LIN {X 0,Y 525.291,Z 461.786,A -85,B 0,C 180,E1 -4783.393,E2 -4783.393} C_VEL
LIN {X 0,Y 525.461,Z 449.021,A -85,B 0,C 180,E1 -4783.659,E2 -4783.659} C_VEL
LIN {X 0,Y 525.774,Z 355.172,A -85,B 0,C 180,E1 -4784.965,E2 -4784.965} C_VEL
LIN {X 0,Y 524.31,Z 344.888,A -85,B 0,C 180,E1 -4785.179,E2 -4785.179} C_VEL
LIN {X 0,Y 524.712,Z 325.315,A -85,B 0,C 180,E1 -4788.014,E2 -4788.014} C_VEL
LIN {X 0,Y 525.255,Z 302.194,A -85,B 0,C 180,E1 -4791.383,E2 -4791.383} C_VEL
LIN {X 0,Y 525.641,Z 284.25,A -85,B 0,C 180,E1 -4794.065,E2 -4794.065} C_VEL
LIN {X 0,Y 523.939,Z 275.222,A -85,B 0,C 180,E1 -4795.549,E2 -4795.549} C_VEL
LIN {X 0,Y 523.92,Z 275.224,A -85,B 0,C 180,E1 -4798.874,E2 -4798.874} C_VEL
LIN {X 0,Y 523.911,Z 275.22,A -85,B 0,C 180,E1 -4801.543,E2 -4801.543} C_VEL
LIN {X 0,Y 523.903,Z 275.225,A -85,B 0,C 180,E1 -4804.29,E2 -4804.29} C_VEL
LIN {X 0,Y 523.871,Z 275.227,A -85,B 0,C 180,E1 -4807.132,E2 -4807.132} C_VEL
LIN {X 0,Y 523.9,Z 275.223,A -85,B 0,C 180,E1 -4810.124,E2 -4810.124} C_VEL
LIN {X 0,Y 523.873,Z 275.226,A -85,B 0,C 180,E1 -4813.168,E2 -4813.168} C_VEL
LIN {X 0,Y 523.907,Z 275.22,A -85,B 0,C 180,E1 -4815.768,E2 -4815.768} C_VEL
LIN {X 0,Y 523.878,Z 275.229,A -85,B 0,C 180,E1 -4818.901,E2 -4818.901} C_VEL
LIN {X 0,Y 523.887,Z 275.223,A -85,B 0,C 180,E1 -4821.895,E2 -4821.895} C_VEL
LIN {X 0,Y 523.895,Z 275.228,A -85,B 0,C 180,E1 -4824.91,E2 -4824.91} C_VEL
LIN {X 0,Y 523.906,Z 275.22,A -85,B 0,C 180,E1 -4827.678,E2 -4827.678} C_VEL
LIN {X 0,Y 523.921,Z 275.226,A -85,B 0,C 180,E1 -4830.675,E2 -4830.675} C_VEL
LIN {X 0,Y 523.909,Z 275.227,A -85,B 0,C 180,E1 -4832.864,E2 -4832.864} C_VEL
LIN {X 0,Y 523.899,Z 275.222,A -85,B 0,C 180,E1 -4835.802,E2 -4835.802} C_VEL
LIN {X 0,Y 523.907,Z 275.228,A -85,B 0,C 180,E1 -4838.765,E2 -4838.765} C_VEL
LIN {X 0,Y 523.902,Z 275.224,A -85,B 0,C 180,E1 -4841.219,E2 -4841.219} C_VEL
LIN {X 0,Y 523.89,Z 275.223,A -85,B 0,C 180,E1 -4843.637,E2 -4843.637} C_VEL
LIN {X 0,Y 523.894,Z 275.223,A -85,B 0,C 180,E1 -4846.026,E2 -4846.026} C_VEL
LIN {X 0,Y 523.975,Z 275.216,A -85,B 0,C 180,E1 -4848.393,E2 -4848.393} C_VEL
LIN {X 0,Y 523.964,Z 275.214,A -85,B 0,C 180,E1 -4851.515,E2 -4851.515} C_VEL
LIN {X 0,Y 524.043,Z 275.21,A -85,B 0,C 180,E1 -4854.613,E2 -4854.613} C_VEL
LIN {X 0,Y 524.066,Z 275.201,A -85,B 0,C 180,E1 -4857.694,E2 -4857.694} C_VEL
LIN {X 0,Y 524.089,Z 275.205,A -85,B 0,C 180,E1 -4860.768,E2 -4860.768} C_VEL
LIN {X 0,Y 524.037,Z 275.21,A -85,B 0,C 180,E1 -4863.075,E2 -4863.075} C_VEL
LIN {X 0,Y 523.997,Z 275.211,A -85,B 0,C 180,E1 -4866.159,E2 -4866.159} C_VEL
LIN {X 0,Y 523.969,Z 275.216,A -85,B 0,C 180,E1 -4869.262,E2 -4869.262} C_VEL
LIN {X 0,Y 523.986,Z 275.211,A -85,B 0,C 180,E1 -4871.752,E2 -4871.752} C_VEL
LIN {X 0,Y 523.954,Z 275.222,A -85,B 0,C 180,E1 -4875.053,E2 -4875.053} C_VEL
LIN {X 0,Y 523.928,Z 275.219,A -85,B 0,C 180,E1 -4877.97,E2 -4877.97} C_VEL
LIN {X 0,Y 523.937,Z 275.22,A -85,B 0,C 180,E1 -4880.411,E2 -4880.411} C_VEL
LIN {X 0,Y 523.881,Z 275.23,A -85,B 0,C 180,E1 -4882.894,E2 -4882.894} C_VEL
LIN {X 0,Y 523.92,Z 275.222,A -85,B 0,C 180,E1 -4885.42,E2 -4885.42} C_VEL
LIN {X 0,Y 523.939,Z 275.217,A -85,B 0,C 180,E1 -4888,E2 -4888} C_VEL
LIN {X 0,Y 523.922,Z 275.225,A -85,B 0,C 180,E1 -4890.858,E2 -4890.858} C_VEL
LIN {X 0,Y 523.934,Z 275.218,A -85,B 0,C 180,E1 -4893.737,E2 -4893.737} C_VEL
LIN {X 0,Y 523.897,Z 275.225,A -85,B 0,C 180,E1 -4896.406,E2 -4896.406} C_VEL
LIN {X 0,Y 523.934,Z 275.224,A -85,B 0,C 180,E1 -4899.083,E2 -4899.083} C_VEL
LIN {X 0,Y 523.934,Z 275.218,A -85,B 0,C 180,E1 -4902.12,E2 -4902.12} C_VEL
LIN {X 0,Y 523.935,Z 275.222,A -85,B 0,C 180,E1 -4905.31,E2 -4905.31} C_VEL
LIN {X 0,Y 523.903,Z 275.227,A -85,B 0,C 180,E1 -4906.94,E2 -4906.94} C_VEL
LIN {X 0,Y 523.24,Z 275.307,A -85,B 0,C 180,E1 -4907.581,E2 -4907.581} C_VEL
LIN {X 0,Y 520.405,Z 275.662,A -85,B 0,C 180,E1 -4908.623,E2 -4908.623} C_VEL
LIN {X 0,Y 518.008,Z 275.959,A -85,B 0,C 180,E1 -4909.462,E2 -4909.462} C_VEL
LIN {X 0,Y 516.978,Z 276.085,A -85,B 0,C 180,E1 -4910.11,E2 -4910.11} C_VEL
LIN {X 0,Y 516.894,Z 276.096,A -85,B 0,C 180,E1 -4910.33,E2 -4910.33} C_VEL
LIN {X 0,Y 516.872,Z 276.101,A -85,B 0,C 180,E1 -4913.343,E2 -4913.343} C_VEL
LIN {X 0,Y 516.898,Z 276.094,A -85,B 0,C 180,E1 -4916.122,E2 -4916.122} C_VEL
LIN {X 0,Y 516.88,Z 276.103,A -85,B 0,C 180,E1 -4918.937,E2 -4918.937} C_VEL
LIN {X 0,Y 516.911,Z 276.094,A -85,B 0,C 180,E1 -4921.586,E2 -4921.586} C_VEL
LIN {X 0,Y 516.923,Z 276.091,A -85,B 0,C 180,E1 -4924.212,E2 -4924.212} C_VEL
LIN {X 0,Y 516.858,Z 276.105,A -85,B 0,C 180,E1 -4926.777,E2 -4926.777} C_VEL
LIN {X 0,Y 516.934,Z 276.09,A -85,B 0,C 180,E1 -4929.732,E2 -4929.732} C_VEL
LIN {X 0,Y 516.925,Z 276.094,A -85,B 0,C 180,E1 -4932.597,E2 -4932.597} C_VEL
LIN {X 0,Y 516.939,Z 276.095,A -85,B 0,C 180,E1 -4935.03,E2 -4935.03} C_VEL
LIN {X 0,Y 516.963,Z 276.086,A -85,B 0,C 180,E1 -4938.234,E2 -4938.234} C_VEL
LIN {X 0,Y 516.967,Z 276.09,A -85,B 0,C 180,E1 -4941.399,E2 -4941.399} C_VEL
LIN {X 0,Y 517.008,Z 276.081,A -85,B 0,C 180,E1 -4943.756,E2 -4943.756} C_VEL
LIN {X 0,Y 517.083,Z 276.073,A -85,B 0,C 180,E1 -4947.662,E2 -4947.662} C_VEL
LIN {X 0,Y 517.09,Z 276.074,A -85,B 0,C 180,E1 -4950.777,E2 -4950.777} C_VEL
LIN {X 0,Y 517.011,Z 276.087,A -85,B 0,C 180,E1 -4953.115,E2 -4953.115} C_VEL
LIN {X 0,Y 516.998,Z 276.081,A -85,B 0,C 180,E1 -4956.241,E2 -4956.241} C_VEL
LIN {X 0,Y 516.947,Z 276.092,A -85,B 0,C 180,E1 -4959.387,E2 -4959.387} C_VEL
LIN {X 0,Y 516.977,Z 276.085,A -85,B 0,C 180,E1 -4961.822,E2 -4961.822} C_VEL
LIN {X 0,Y 516.935,Z 276.096,A -85,B 0,C 180,E1 -4965.144,E2 -4965.144} C_VEL
LIN {X 0,Y 516.915,Z 276.091,A -85,B 0,C 180,E1 -4968.219,E2 -4968.219} C_VEL
LIN {X 0,Y 516.903,Z 276.095,A -85,B 0,C 180,E1 -4970.698,E2 -4970.698} C_VEL
LIN {X 0,Y 516.877,Z 276.103,A -85,B 0,C 180,E1 -4973.219,E2 -4973.219} C_VEL
LIN {X 0,Y 516.928,Z 276.089,A -85,B 0,C 180,E1 -4976.194,E2 -4976.194} C_VEL
LIN {X 0,Y 516.916,Z 276.098,A -85,B 0,C 180,E1 -4979.3,E2 -4979.3} C_VEL
LIN {X 0,Y 516.881,Z 276.096,A -85,B 0,C 180,E1 -4982.541,E2 -4982.541} C_VEL
LIN {X 0,Y 516.858,Z 276.105,A -85,B 0,C 180,E1 -4985.329,E2 -4985.329} C_VEL
LIN {X 0,Y 516.858,Z 276.098,A -85,B 0,C 180,E1 -4987.941,E2 -4987.941} C_VEL
LIN {X 0,Y 516.886,Z 276.098,A -85,B 0,C 180,E1 -4990.735,E2 -4990.735} C_VEL
LIN {X 0,Y 517.02,Z 276.175,A -85,B 0,C 180,E1 -4993.84,E2 -4993.84} C_VEL
LIN {X 0,Y 517.32,Z 280.633,A -85,B 0,C 180,E1 -4994.754,E2 -4994.754} C_VEL
LIN {X 0,Y 517.177,Z 290.379,A -85,B 0,C 180,E1 -4996.7,E2 -4996.7} C_VEL
LIN {X 0,Y 519.112,Z 300.838,A -85,B 0,C 180,E1 -4996.916,E2 -4996.916} C_VEL
LIN {X 0,Y 518.557,Z 397.529,A -85,B 0,C 180,E1 -4998.312,E2 -4998.312} C_VEL
LIN {X 0,Y 518.413,Z 410.717,A -85,B 0,C 180,E1 -4998.665,E2 -4998.665} C_VEL
LIN {X 0,Y 518.158,Z 422.479,A -85,B 0,C 180,E1 -4999.124,E2 -4999.124} C_VEL
LIN {X 0,Y 517.938,Z 434.251,A -85,B 0,C 180,E1 -4999.742,E2 -4999.742} C_VEL
LIN {X 0,Y 517.615,Z 444.905,A -85,B 0,C 180,E1 -5000.459,E2 -5000.459} C_VEL
LIN {X 0,Y 517.342,Z 455.25,A -85,B 0,C 180,E1 -5001.326,E2 -5001.326} C_VEL
LIN {X 0,Y 517.089,Z 464.659,A -85,B 0,C 180,E1 -5002.294,E2 -5002.294} C_VEL
LIN {X 0,Y 516.852,Z 472.928,A -85,B 0,C 180,E1 -5003.337,E2 -5003.337} C_VEL
LIN {X 0,Y 516.659,Z 480.32,A -85,B 0,C 180,E1 -5004.488,E2 -5004.488} C_VEL
LIN {X 0,Y 516.517,Z 486.204,A -85,B 0,C 180,E1 -5005.621,E2 -5005.621} C_VEL
LIN {X 0,Y 516.373,Z 491.862,A -85,B 0,C 180,E1 -5007.016,E2 -5007.016} C_VEL
LIN {X 0,Y 516.34,Z 495.956,A -85,B 0,C 180,E1 -5008.398,E2 -5008.398} C_VEL
LIN {X 0,Y 516.238,Z 498.614,A -85,B 0,C 180,E1 -5009.755,E2 -5009.755} C_VEL
LIN {X 0,Y 516.205,Z 499.695,A -85,B 0,C 180,E1 -5010.651,E2 -5010.651} C_VEL
LIN {X 0,Y 516.199,Z 500.248,A -85,B 0,C 180,E1 -5011.542,E2 -5011.542} C_VEL
LIN {X 0,Y 516.168,Z 500.291,A -85,B 0,C 180,E1 -5012.424,E2 -5012.424} C_VEL
LIN {X 0,Y 516.187,Z 499.855,A -85,B 0,C 180,E1 -5013.302,E2 -5013.302} C_VEL
LIN {X 0,Y 516.226,Z 498.881,A -85,B 0,C 180,E1 -5014.174,E2 -5014.174} C_VEL
LIN {X 0,Y 516.272,Z 497.427,A -85,B 0,C 180,E1 -5015.039,E2 -5015.039} C_VEL
LIN {X 0,Y 516.4,Z 494.312,A -85,B 0,C 180,E1 -5016.33,E2 -5016.33} C_VEL
LIN {X 0,Y 516.455,Z 489.615,A -85,B 0,C 180,E1 -5017.704,E2 -5017.704} C_VEL
LIN {X 0,Y 516.569,Z 483.336,A -85,B 0,C 180,E1 -5019.076,E2 -5019.076} C_VEL
LIN {X 0,Y 516.801,Z 475.952,A -85,B 0,C 180,E1 -5020.332,E2 -5020.332} C_VEL
LIN {X 0,Y 516.981,Z 468.38,A -85,B 0,C 180,E1 -5021.37,E2 -5021.37} C_VEL
LIN {X 0,Y 517.287,Z 458.631,A -85,B 0,C 180,E1 -5022.455,E2 -5022.455} C_VEL
LIN {X 0,Y 517.533,Z 448.953,A -85,B 0,C 180,E1 -5023.33,E2 -5023.33} C_VEL
LIN {X 0,Y 517.863,Z 437.568,A -85,B 0,C 180,E1 -5024.15,E2 -5024.15} C_VEL
LIN {X 0,Y 518.14,Z 425.417,A -85,B 0,C 180,E1 -5024.832,E2 -5024.832} C_VEL
LIN {X 0,Y 518.303,Z 413.887,A -85,B 0,C 180,E1 -5025.322,E2 -5025.322} C_VEL
LIN {X 0,Y 518.48,Z 401.522,A -85,B 0,C 180,E1 -5025.69,E2 -5025.69} C_VEL
LIN {X 0,Y 518.625,Z 386.132,A -85,B 0,C 180,E1 -5025.957,E2 -5025.957} C_VEL
LIN {X 0,Y 519.014,Z 299.941,A -85,B 0,C 180,E1 -5027.195,E2 -5027.195} C_VEL
LIN {X 0,Y 517.1,Z 289.663,A -85,B 0,C 180,E1 -5027.42,E2 -5027.42} C_VEL
LIN {X 0,Y 516.929,Z 276.096,A -85,B 0,C 180,E1 -5029.622,E2 -5029.622} C_VEL
LIN {X 0,Y 516.953,Z 276.095,A -85,B 0,C 180,E1 -5032.972,E2 -5032.972} C_VEL
LIN {X 0,Y 516.877,Z 276.102,A -85,B 0,C 180,E1 -5035.321,E2 -5035.321} C_VEL
LIN {X 0,Y 517.021,Z 276.081,A -85,B 0,C 180,E1 -5037.663,E2 -5037.663} C_VEL
LIN {X 0,Y 517.038,Z 276.083,A -85,B 0,C 180,E1 -5040.779,E2 -5040.779} C_VEL
LIN {X 0,Y 516.987,Z 276.09,A -85,B 0,C 180,E1 -5043.117,E2 -5043.117} C_VEL
LIN {X 0,Y 516.95,Z 276.088,A -85,B 0,C 180,E1 -5046.244,E2 -5046.244} C_VEL
LIN {X 0,Y 516.906,Z 276.096,A -85,B 0,C 180,E1 -5049.39,E2 -5049.39} C_VEL
LIN {X 0,Y 516.925,Z 276.09,A -85,B 0,C 180,E1 -5051.826,E2 -5051.826} C_VEL
LIN {X 0,Y 516.899,Z 276.1,A -85,B 0,C 180,E1 -5055.154,E2 -5055.154} C_VEL
LIN {X 0,Y 516.872,Z 276.095,A -85,B 0,C 180,E1 -5058.225,E2 -5058.225} C_VEL
LIN {X 0,Y 516.859,Z 276.1,A -85,B 0,C 180,E1 -5060.704,E2 -5060.704} C_VEL
LIN {X 0,Y 516.86,Z 276.098,A -85,B 0,C 180,E1 -5064.075,E2 -5064.075} C_VEL
LIN {X 0,Y 516.88,Z 276.096,A -85,B 0,C 180,E1 -5066.661,E2 -5066.661} C_VEL
LIN {X 0,Y 516.863,Z 276.101,A -85,B 0,C 180,E1 -5069.527,E2 -5069.527} C_VEL
LIN {X 0,Y 516.856,Z 276.099,A -85,B 0,C 180,E1 -5072.548,E2 -5072.548} C_VEL
LIN {X 0,Y 516.84,Z 276.108,A -85,B 0,C 180,E1 -5075.336,E2 -5075.336} C_VEL
LIN {X 0,Y 516.841,Z 276.101,A -85,B 0,C 180,E1 -5077.947,E2 -5077.947} C_VEL
LIN {X 0,Y 516.872,Z 276.098,A -85,B 0,C 180,E1 -5080.743,E2 -5080.743} C_VEL
LIN {X 0,Y 516.849,Z 276.1,A -85,B 0,C 180,E1 -5083.907,E2 -5083.907} C_VEL
LIN {X 0,Y 516.852,Z 276.099,A -85,B 0,C 180,E1 -5086.111,E2 -5086.111} C_VEL
LIN {X 0,Y 516.888,Z 276.095,A -85,B 0,C 180,E1 -5088.402,E2 -5088.402} C_VEL
LIN {X 0,Y 516.854,Z 276.107,A -85,B 0,C 180,E1 -5091.288,E2 -5091.288} C_VEL
LIN {X 0,Y 516.848,Z 276.101,A -85,B 0,C 180,E1 -5094.224,E2 -5094.224} C_VEL
LIN {X 0,Y 516.875,Z 276.105,A -85,B 0,C 180,E1 -5097.057,E2 -5097.057} C_VEL
LIN {X 0,Y 516.875,Z 276.103,A -85,B 0,C 180,E1 -5099.8,E2 -5099.8} C_VEL
LIN {X 0,Y 516.886,Z 276.097,A -85,B 0,C 180,E1 -5102.469,E2 -5102.469} C_VEL
LIN {X 0,Y 516.983,Z 276.197,A -85,B 0,C 180,E1 -5104.892,E2 -5104.892} C_VEL
LIN {X 0,Y 518.182,Z 283.513,A -85,B 0,C 180,E1 -5105.995,E2 -5105.995} C_VEL
LIN {X 0,Y 518.031,Z 299.695,A -85,B 0,C 180,E1 -5108.307,E2 -5108.307} C_VEL
LIN {X 0,Y 517.64,Z 321.277,A -85,B 0,C 180,E1 -5111.397,E2 -5111.397} C_VEL
LIN {X 0,Y 517.269,Z 343.187,A -85,B 0,C 180,E1 -5114.518,E2 -5114.518} C_VEL
LIN {X 0,Y 517.262,Z 343.958,A -85,B 0,C 180,E1 -5114.627,E2 -5114.627} C_VEL
LIN {X 0,Y 519.01,Z 357.136,A -85,B 0,C 180,E1 -5114.877,E2 -5114.877} C_VEL
LIN {X 0,Y 518.494,Z 453.268,A -85,B 0,C 180,E1 -5116.256,E2 -5116.256} C_VEL
LIN {X 0,Y 518.213,Z 467.238,A -85,B 0,C 180,E1 -5116.623,E2 -5116.623} C_VEL
LIN {X 0,Y 517.945,Z 479.777,A -85,B 0,C 180,E1 -5117.115,E2 -5117.115} C_VEL
LIN {X 0,Y 517.687,Z 492.67,A -85,B 0,C 180,E1 -5117.812,E2 -5117.812} C_VEL
LIN {X 0,Y 517.38,Z 504.601,A -85,B 0,C 180,E1 -5118.643,E2 -5118.643} C_VEL
LIN {X 0,Y 517.132,Z 513.696,A -85,B 0,C 180,E1 -5119.43,E2 -5119.43} C_VEL
LIN {X 0,Y 516.862,Z 523.026,A -85,B 0,C 180,E1 -5120.414,E2 -5120.414} C_VEL
LIN {X 0,Y 516.643,Z 532.102,A -85,B 0,C 180,E1 -5121.593,E2 -5121.593} C_VEL
LIN {X 0,Y 516.503,Z 539.416,A -85,B 0,C 180,E1 -5122.771,E2 -5122.771} C_VEL
LIN {X 0,Y 516.389,Z 544.343,A -85,B 0,C 180,E1 -5123.751,E2 -5123.751} C_VEL
LIN {X 0,Y 516.312,Z 549.136,A -85,B 0,C 180,E1 -5124.926,E2 -5124.926} C_VEL
LIN {X 0,Y 516.37,Z 552.805,A -85,B 0,C 180,E1 -5126.1,E2 -5126.1} C_VEL
LIN {X 0,Y 516.282,Z 554.693,A -85,B 0,C 180,E1 -5126.88,E2 -5126.88} C_VEL
LIN {X 0,Y 516.261,Z 556.11,A -85,B 0,C 180,E1 -5127.661,E2 -5127.661} C_VEL
LIN {X 0,Y 516.168,Z 557.737,A -85,B 0,C 180,E1 -5129.221,E2 -5129.221} C_VEL
LIN {X 0,Y 516.17,Z 557.962,A -85,B 0,C 180,E1 -5130.001,E2 -5130.001} C_VEL
LIN {X 0,Y 516.192,Z 557.138,A -85,B 0,C 180,E1 -5131.561,E2 -5131.561} C_VEL
LIN {X 0,Y 516.261,Z 556.14,A -85,B 0,C 180,E1 -5132.342,E2 -5132.342} C_VEL
LIN {X 0,Y 516.283,Z 554.732,A -85,B 0,C 180,E1 -5133.122,E2 -5133.122} C_VEL
LIN {X 0,Y 516.313,Z 551.77,A -85,B 0,C 180,E1 -5134.294,E2 -5134.294} C_VEL
LIN {X 0,Y 516.397,Z 547.759,A -85,B 0,C 180,E1 -5135.467,E2 -5135.467} C_VEL
LIN {X 0,Y 516.452,Z 541.783,A -85,B 0,C 180,E1 -5136.8,E2 -5136.8} C_VEL
LIN {X 0,Y 516.585,Z 534.83,A -85,B 0,C 180,E1 -5138.016,E2 -5138.016} C_VEL
LIN {X 0,Y 516.771,Z 526.454,A -85,B 0,C 180,E1 -5139.195,E2 -5139.195} C_VEL
LIN {X 0,Y 517.004,Z 517.847,A -85,B 0,C 180,E1 -5140.179,E2 -5140.179} C_VEL
LIN {X 0,Y 517.349,Z 507.228,A -85,B 0,C 180,E1 -5141.162,E2 -5141.162} C_VEL
LIN {X 0,Y 517.652,Z 495.942,A -85,B 0,C 180,E1 -5142.002,E2 -5142.002} C_VEL
LIN {X 0,Y 517.92,Z 485.132,A -85,B 0,C 180,E1 -5142.639,E2 -5142.639} C_VEL
LIN {X 0,Y 518.164,Z 473.127,A -85,B 0,C 180,E1 -5143.181,E2 -5143.181} C_VEL
LIN {X 0,Y 518.406,Z 460.182,A -85,B 0,C 180,E1 -5143.599,E2 -5143.599} C_VEL
LIN {X 0,Y 518.573,Z 446.517,A -85,B 0,C 180,E1 -5143.869,E2 -5143.869} C_VEL
LIN {X 0,Y 518.906,Z 355.844,A -85,B 0,C 180,E1 -5145.152,E2 -5145.152} C_VEL
LIN {X 0,Y 517.308,Z 344.698,A -85,B 0,C 180,E1 -5145.365,E2 -5145.365} C_VEL
LIN {X 0,Y 517.726,Z 325.447,A -85,B 0,C 180,E1 -5148.192,E2 -5148.192} C_VEL
LIN {X 0,Y 518.308,Z 303.272,A -85,B 0,C 180,E1 -5151.475,E2 -5151.475} C_VEL
LIN {X 0,Y 518.704,Z 285.555,A -85,B 0,C 180,E1 -5154.163,E2 -5154.163} C_VEL
LIN {X 0,Y 516.884,Z 276.101,A -85,B 0,C 180,E1 -5155.736,E2 -5155.736} C_VEL
LIN {X 0,Y 516.855,Z 276.106,A -85,B 0,C 180,E1 -5158.417,E2 -5158.417} C_VEL
LIN {X 0,Y 516.88,Z 276.098,A -85,B 0,C 180,E1 -5161.108,E2 -5161.108} C_VEL
LIN {X 0,Y 516.872,Z 276.097,A -85,B 0,C 180,E1 -5163.96,E2 -5163.96} C_VEL
LIN {X 0,Y 516.833,Z 276.109,A -85,B 0,C 180,E1 -5166.747,E2 -5166.747} C_VEL
LIN {X 0,Y 516.845,Z 276.1,A -85,B 0,C 180,E1 -5169.722,E2 -5169.722} C_VEL
LIN {X 0,Y 516.868,Z 276.097,A -85,B 0,C 180,E1 -5171.776,E2 -5171.776} C_VEL
LIN {X 0,Y 516.879,Z 276.1,A -85,B 0,C 180,E1 -5175.005,E2 -5175.005} C_VEL
LIN {X 0,Y 516.867,Z 276.102,A -85,B 0,C 180,E1 -5178.4,E2 -5178.4} C_VEL
LIN {X 0,Y 516.854,Z 276.1,A -85,B 0,C 180,E1 -5181.281,E2 -5181.281} C_VEL
LIN {X 0,Y 516.841,Z 276.103,A -85,B 0,C 180,E1 -5184.217,E2 -5184.217} C_VEL
LIN {X 0,Y 516.854,Z 276.103,A -85,B 0,C 180,E1 -5187.05,E2 -5187.05} C_VEL
LIN {X 0,Y 516.853,Z 276.099,A -85,B 0,C 180,E1 -5189.793,E2 -5189.793} C_VEL
LIN {X 0,Y 516.889,Z 276.1,A -85,B 0,C 180,E1 -5192.465,E2 -5192.465} C_VEL
LIN {X 0,Y 516.838,Z 276.101,A -85,B 0,C 180,E1 -5195.644,E2 -5195.644} C_VEL
LIN {X 0,Y 516.848,Z 276.105,A -85,B 0,C 180,E1 -5198.46,E2 -5198.46} C_VEL
LIN {X 0,Y 516.855,Z 276.105,A -85,B 0,C 180,E1 -5200.953,E2 -5200.953} C_VEL
LIN {X 0,Y 516.865,Z 276.099,A -85,B 0,C 180,E1 -5203.408,E2 -5203.408} C_VEL
LIN {X 0,Y 516.85,Z 276.1,A -85,B 0,C 180,E1 -5205.832,E2 -5205.832} C_VEL
LIN {X 0,Y 516.968,Z 276.087,A -85,B 0,C 180,E1 -5208.233,E2 -5208.233} C_VEL
LIN {X 0,Y 516.93,Z 276.091,A -85,B 0,C 180,E1 -5211.399,E2 -5211.399} C_VEL
LIN {X 0,Y 516.963,Z 276.086,A -85,B 0,C 180,E1 -5213.756,E2 -5213.756} C_VEL
LIN {X 0,Y 516.977,Z 276.091,A -85,B 0,C 180,E1 -5216.882,E2 -5216.882} C_VEL
LIN {X 0,Y 517.038,Z 276.077,A -85,B 0,C 180,E1 -5220,E2 -5220} C_VEL
LIN {X 0,Y 516.978,Z 276.089,A -85,B 0,C 180,E1 -5223.117,E2 -5223.117} C_VEL
LIN {X 0,Y 516.962,Z 276.088,A -85,B 0,C 180,E1 -5226.243,E2 -5226.243} C_VEL
LIN {X 0,Y 516.924,Z 276.093,A -85,B 0,C 180,E1 -5229.389,E2 -5229.389} C_VEL
LIN {X 0,Y 516.945,Z 276.088,A -85,B 0,C 180,E1 -5231.825,E2 -5231.825} C_VEL
LIN {X 0,Y 516.905,Z 276.098,A -85,B 0,C 180,E1 -5235.146,E2 -5235.146} C_VEL
LIN {X 0,Y 516.89,Z 276.097,A -85,B 0,C 180,E1 -5238.223,E2 -5238.223} C_VEL
LIN {X 0,Y 516.877,Z 276.103,A -85,B 0,C 180,E1 -5240.702,E2 -5240.702} C_VEL
LIN {X 0,Y 516.877,Z 276.097,A -85,B 0,C 180,E1 -5244.073,E2 -5244.073} C_VEL
LIN {X 0,Y 516.896,Z 276.1,A -85,B 0,C 180,E1 -5246.659,E2 -5246.659} C_VEL
LIN {X 0,Y 516.893,Z 276.096,A -85,B 0,C 180,E1 -5249.528,E2 -5249.528} C_VEL
LIN {X 0,Y 516.871,Z 276.102,A -85,B 0,C 180,E1 -5252.546,E2 -5252.546} C_VEL
LIN {X 0,Y 516.856,Z 276.103,A -85,B 0,C 180,E1 -5255.334,E2 -5255.334} C_VEL
LIN {X 0,Y 516.856,Z 276.1,A -85,B 0,C 180,E1 -5257.945,E2 -5257.945} C_VEL
LIN {X 0,Y 516.881,Z 276.103,A -85,B 0,C 180,E1 -5260.741,E2 -5260.741} C_VEL
LIN {X 0,Y 516.861,Z 276.099,A -85,B 0,C 180,E1 -5263.905,E2 -5263.905} C_VEL
LIN {X 0,Y 516.863,Z 276.099,A -85,B 0,C 180,E1 -5266.109,E2 -5266.109} C_VEL
LIN {X 0,Y 516.888,Z 276.1,A -85,B 0,C 180,E1 -5269.262,E2 -5269.262} C_VEL
LIN {X 0,Y 516.894,Z 276.096,A -85,B 0,C 180,E1 -5270.33,E2 -5270.33} C_VEL
LIN {X 0,Y 516.226,Z 276.184,A -85,B 0,C 180,E1 -5270.98,E2 -5270.98} C_VEL
LIN {X 0,Y 513.369,Z 276.54,A -85,B 0,C 180,E1 -5272.035,E2 -5272.035} C_VEL
LIN {X 0,Y 510.95,Z 276.841,A -85,B 0,C 180,E1 -5272.885,E2 -5272.885} C_VEL
LIN {X 0,Y 509.906,Z 276.968,A -85,B 0,C 180,E1 -5273.542,E2 -5273.542} C_VEL
LIN {X 0,Y 509.818,Z 276.977,A -85,B 0,C 180,E1 -5273.764,E2 -5273.764} C_VEL
LIN {X 0,Y 509.848,Z 276.976,A -85,B 0,C 180,E1 -5276.541,E2 -5276.541} C_VEL
LIN {X 0,Y 509.834,Z 276.979,A -85,B 0,C 180,E1 -5279.335,E2 -5279.335} C_VEL
LIN {X 0,Y 509.885,Z 276.968,A -85,B 0,C 180,E1 -5282.056,E2 -5282.056} C_VEL
LIN {X 0,Y 509.868,Z 276.975,A -85,B 0,C 180,E1 -5284.705,E2 -5284.705} C_VEL
LIN {X 0,Y 509.82,Z 276.979,A -85,B 0,C 180,E1 -5287.459,E2 -5287.459} C_VEL
LIN {X 0,Y 509.912,Z 276.965,A -85,B 0,C 180,E1 -5289.845,E2 -5289.845} C_VEL
LIN {X 0,Y 509.88,Z 276.973,A -85,B 0,C 180,E1 -5293.175,E2 -5293.175} C_VEL
LIN {X 0,Y 509.86,Z 276.973,A -85,B 0,C 180,E1 -5295.634,E2 -5295.634} C_VEL
LIN {X 0,Y 509.91,Z 276.971,A -85,B 0,C 180,E1 -5298.874,E2 -5298.874} C_VEL
LIN {X 0,Y 509.95,Z 276.96,A -85,B 0,C 180,E1 -5302.078,E2 -5302.078} C_VEL
LIN {X 0,Y 509.979,Z 276.957,A -85,B 0,C 180,E1 -5304.464,E2 -5304.464} C_VEL
LIN {X 0,Y 510.053,Z 276.949,A -85,B 0,C 180,E1 -5307.63,E2 -5307.63} C_VEL
LIN {X 0,Y 510.061,Z 276.95,A -85,B 0,C 180,E1 -5310.788,E2 -5310.788} C_VEL
LIN {X 0,Y 509.953,Z 276.965,A -85,B 0,C 180,E1 -5313.159,E2 -5313.159} C_VEL
LIN {X 0,Y 509.949,Z 276.96,A -85,B 0,C 180,E1 -5316.328,E2 -5316.328} C_VEL
LIN {X 0,Y 509.91,Z 276.968,A -85,B 0,C 180,E1 -5318.718,E2 -5318.718} C_VEL
LIN {X 0,Y 509.944,Z 276.96,A -85,B 0,C 180,E1 -5321.928,E2 -5321.928} C_VEL
LIN {X 0,Y 509.885,Z 276.973,A -85,B 0,C 180,E1 -5325.239,E2 -5325.239} C_VEL
LIN {X 0,Y 509.878,Z 276.968,A -85,B 0,C 180,E1 -5327.998,E2 -5327.998} C_VEL
LIN {X 0,Y 509.845,Z 276.979,A -85,B 0,C 180,E1 -5330.998,E2 -5330.998} C_VEL
LIN {X 0,Y 509.836,Z 276.976,A -85,B 0,C 180,E1 -5333.559,E2 -5333.559} C_VEL
LIN {X 0,Y 509.897,Z 276.966,A -85,B 0,C 180,E1 -5336.376,E2 -5336.376} C_VEL
LIN {X 0,Y 509.866,Z 276.973,A -85,B 0,C 180,E1 -5338.84,E2 -5338.84} C_VEL
LIN {X 0,Y 509.805,Z 276.98,A -85,B 0,C 180,E1 -5341.586,E2 -5341.586} C_VEL
LIN {X 0,Y 509.83,Z 276.974,A -85,B 0,C 180,E1 -5344.41,E2 -5344.41} C_VEL
LIN {X 0,Y 509.795,Z 276.986,A -85,B 0,C 180,E1 -5347.337,E2 -5347.337} C_VEL
LIN {X 0,Y 509.848,Z 276.973,A -85,B 0,C 180,E1 -5350.375,E2 -5350.375} C_VEL
LIN {X 0,Y 509.961,Z 277.14,A -85,B 0,C 180,E1 -5353.746,E2 -5353.746} C_VEL
LIN {X 0,Y 510.361,Z 281.307,A -85,B 0,C 180,E1 -5354.604,E2 -5354.604} C_VEL
LIN {X 0,Y 510.193,Z 290.656,A -85,B 0,C 180,E1 -5356.48,E2 -5356.48} C_VEL
LIN {X 0,Y 512.285,Z 302.196,A -85,B 0,C 180,E1 -5356.725,E2 -5356.725} C_VEL
LIN {X 0,Y 511.655,Z 397.696,A -85,B 0,C 180,E1 -5358.128,E2 -5358.128} C_VEL
LIN {X 0,Y 511.525,Z 411.164,A -85,B 0,C 180,E1 -5358.494,E2 -5358.494} C_VEL
LIN {X 0,Y 511.24,Z 423.429,A -85,B 0,C 180,E1 -5358.982,E2 -5358.982} C_VEL
LIN {X 0,Y 510.985,Z 435.16,A -85,B 0,C 180,E1 -5359.617,E2 -5359.617} C_VEL
LIN {X 0,Y 510.654,Z 445.366,A -85,B 0,C 180,E1 -5360.316,E2 -5360.316} C_VEL
LIN {X 0,Y 510.357,Z 455.802,A -85,B 0,C 180,E1 -5361.203,E2 -5361.203} C_VEL
LIN {X 0,Y 510.094,Z 465.191,A -85,B 0,C 180,E1 -5362.186,E2 -5362.186} C_VEL
LIN {X 0,Y 509.822,Z 474.192,A -85,B 0,C 180,E1 -5363.356,E2 -5363.356} C_VEL
LIN {X 0,Y 509.567,Z 481.882,A -85,B 0,C 180,E1 -5364.601,E2 -5364.601} C_VEL
LIN {X 0,Y 509.435,Z 488.033,A -85,B 0,C 180,E1 -5365.857,E2 -5365.857} C_VEL
LIN {X 0,Y 509.327,Z 492.216,A -85,B 0,C 180,E1 -5366.94,E2 -5366.94} C_VEL
LIN {X 0,Y 509.265,Z 496.387,A -85,B 0,C 180,E1 -5368.372,E2 -5368.372} C_VEL
LIN {X 0,Y 509.177,Z 498.288,A -85,B 0,C 180,E1 -5369.29,E2 -5369.29} C_VEL
LIN {X 0,Y 509.132,Z 499.858,A -85,B 0,C 180,E1 -5370.405,E2 -5370.405} C_VEL
LIN {X 0,Y 509.106,Z 500.75,A -85,B 0,C 180,E1 -5372.008,E2 -5372.008} C_VEL
LIN {X 0,Y 509.094,Z 500.509,A -85,B 0,C 180,E1 -5372.899,E2 -5372.899} C_VEL
LIN {X 0,Y 509.143,Z 499.791,A -85,B 0,C 180,E1 -5373.787,E2 -5373.787} C_VEL
LIN {X 0,Y 509.173,Z 498.585,A -85,B 0,C 180,E1 -5374.667,E2 -5374.667} C_VEL
LIN {X 0,Y 509.269,Z 495.719,A -85,B 0,C 180,E1 -5376.014,E2 -5376.014} C_VEL
LIN {X 0,Y 509.366,Z 491.881,A -85,B 0,C 180,E1 -5377.274,E2 -5377.274} C_VEL
LIN {X 0,Y 509.472,Z 486.694,A -85,B 0,C 180,E1 -5378.558,E2 -5378.558} C_VEL
LIN {X 0,Y 509.693,Z 480.084,A -85,B 0,C 180,E1 -5379.836,E2 -5379.836} C_VEL
LIN {X 0,Y 509.875,Z 471.759,A -85,B 0,C 180,E1 -5381.1,E2 -5381.1} C_VEL
LIN {X 0,Y 510.24,Z 462.302,A -85,B 0,C 180,E1 -5382.249,E2 -5382.249} C_VEL
LIN {X 0,Y 510.473,Z 452.647,A -85,B 0,C 180,E1 -5383.195,E2 -5383.195} C_VEL
LIN {X 0,Y 510.848,Z 441.043,A -85,B 0,C 180,E1 -5384.101,E2 -5384.101} C_VEL
LIN {X 0,Y 511.101,Z 429.877,A -85,B 0,C 180,E1 -5384.791,E2 -5384.791} C_VEL
LIN {X 0,Y 511.349,Z 417.436,A -85,B 0,C 180,E1 -5385.372,E2 -5385.372} C_VEL
LIN {X 0,Y 511.549,Z 404.165,A -85,B 0,C 180,E1 -5385.81,E2 -5385.81} C_VEL
LIN {X 0,Y 511.737,Z 391.341,A -85,B 0,C 180,E1 -5386.069,E2 -5386.069} C_VEL
LIN {X 0,Y 512.179,Z 300.819,A -85,B 0,C 180,E1 -5387.394,E2 -5387.394} C_VEL
LIN {X 0,Y 510.162,Z 289.959,A -85,B 0,C 180,E1 -5387.646,E2 -5387.646} C_VEL
LIN {X 0,Y 509.878,Z 276.989,A -85,B 0,C 180,E1 -5389.703,E2 -5389.703} C_VEL
LIN {X 0,Y 509.931,Z 276.97,A -85,B 0,C 180,E1 -5392.875,E2 -5392.875} C_VEL
LIN {X 0,Y 509.846,Z 276.979,A -85,B 0,C 180,E1 -5395.256,E2 -5395.256} C_VEL
LIN {X 0,Y 509.994,Z 276.957,A -85,B 0,C 180,E1 -5397.631,E2 -5397.631} C_VEL
LIN {X 0,Y 510.008,Z 276.959,A -85,B 0,C 180,E1 -5400.79,E2 -5400.79} C_VEL
LIN {X 0,Y 509.927,Z 276.969,A -85,B 0,C 180,E1 -5403.161,E2 -5403.161} C_VEL
LIN {X 0,Y 509.918,Z 276.964,A -85,B 0,C 180,E1 -5406.331,E2 -5406.331} C_VEL
LIN {X 0,Y 509.862,Z 276.975,A -85,B 0,C 180,E1 -5408.722,E2 -5408.722} C_VEL
LIN {X 0,Y 509.893,Z 276.966,A -85,B 0,C 180,E1 -5411.932,E2 -5411.932} C_VEL
LIN {X 0,Y 509.844,Z 276.978,A -85,B 0,C 180,E1 -5415.247,E2 -5415.247} C_VEL
LIN {X 0,Y 509.833,Z 276.972,A -85,B 0,C 180,E1 -5418.003,E2 -5418.003} C_VEL
LIN {X 0,Y 509.797,Z 276.983,A -85,B 0,C 180,E1 -5421.004,E2 -5421.004} C_VEL
LIN {X 0,Y 509.819,Z 276.976,A -85,B 0,C 180,E1 -5424.429,E2 -5424.429} C_VEL
LIN {X 0,Y 509.839,Z 276.979,A -85,B 0,C 180,E1 -5427.059,E2 -5427.059} C_VEL
LIN {X 0,Y 509.811,Z 276.978,A -85,B 0,C 180,E1 -5429.754,E2 -5429.754} C_VEL
LIN {X 0,Y 509.833,Z 276.976,A -85,B 0,C 180,E1 -5432.778,E2 -5432.778} C_VEL
LIN {X 0,Y 509.799,Z 276.981,A -85,B 0,C 180,E1 -5435.584,E2 -5435.584} C_VEL
LIN {X 0,Y 509.813,Z 276.976,A -85,B 0,C 180,E1 -5438.342,E2 -5438.342} C_VEL
LIN {X 0,Y 509.835,Z 276.978,A -85,B 0,C 180,E1 -5441.428,E2 -5441.428} C_VEL
LIN {X 0,Y 509.825,Z 276.976,A -85,B 0,C 180,E1 -5444.672,E2 -5444.672} C_VEL
LIN {X 0,Y 509.83,Z 276.974,A -85,B 0,C 180,E1 -5448.107,E2 -5448.107} C_VEL
LIN {X 0,Y 509.82,Z 276.976,A -85,B 0,C 180,E1 -5450.651,E2 -5450.651} C_VEL
LIN {X 0,Y 509.802,Z 276.984,A -85,B 0,C 180,E1 -5453.651,E2 -5453.651} C_VEL
LIN {X 0,Y 509.839,Z 276.977,A -85,B 0,C 180,E1 -5456.543,E2 -5456.543} C_VEL
LIN {X 0,Y 509.828,Z 276.986,A -85,B 0,C 180,E1 -5459.338,E2 -5459.338} C_VEL
LIN {X 0,Y 509.84,Z 276.976,A -85,B 0,C 180,E1 -5462.056,E2 -5462.056} C_VEL
LIN {X 0,Y 509.955,Z 277.151,A -85,B 0,C 180,E1 -5464.758,E2 -5464.758} C_VEL
LIN {X 0,Y 511.171,Z 284.329,A -85,B 0,C 180,E1 -5465.86,E2 -5465.86} C_VEL
LIN {X 0,Y 511.087,Z 296.079,A -85,B 0,C 180,E1 -5467.571,E2 -5467.571} C_VEL
LIN {X 0,Y 510.768,Z 313.524,A -85,B 0,C 180,E1 -5470.093,E2 -5470.093} C_VEL
LIN {X 0,Y 510.429,Z 333.636,A -85,B 0,C 180,E1 -5472.99,E2 -5472.99} C_VEL
LIN {X 0,Y 510.237,Z 343.672,A -85,B 0,C 180,E1 -5474.417,E2 -5474.417} C_VEL
LIN {X 0,Y 512.161,Z 357.72,A -85,B 0,C 180,E1 -5474.685,E2 -5474.685} C_VEL
LIN {X 0,Y 511.579,Z 453.492,A -85,B 0,C 180,E1 -5476.092,E2 -5476.092} C_VEL
LIN {X 0,Y 511.274,Z 467.232,A -85,B 0,C 180,E1 -5476.463,E2 -5476.463} C_VEL
LIN {X 0,Y 510.961,Z 480.142,A -85,B 0,C 180,E1 -5476.986,E2 -5476.986} C_VEL
LIN {X 0,Y 510.719,Z 491.859,A -85,B 0,C 180,E1 -5477.63,E2 -5477.63} C_VEL
LIN {X 0,Y 510.364,Z 504.035,A -85,B 0,C 180,E1 -5478.485,E2 -5478.485} C_VEL
LIN {X 0,Y 510.113,Z 513.162,A -85,B 0,C 180,E1 -5479.283,E2 -5479.283} C_VEL
LIN {X 0,Y 509.817,Z 522.522,A -85,B 0,C 180,E1 -5480.28,E2 -5480.28} C_VEL
LIN {X 0,Y 509.581,Z 531.622,A -85,B 0,C 180,E1 -5481.476,E2 -5481.476} C_VEL
LIN {X 0,Y 509.425,Z 538.956,A -85,B 0,C 180,E1 -5482.67,E2 -5482.67} C_VEL
LIN {X 0,Y 509.307,Z 543.899,A -85,B 0,C 180,E1 -5483.664,E2 -5483.664} C_VEL
LIN {X 0,Y 509.246,Z 548.708,A -85,B 0,C 180,E1 -5484.855,E2 -5484.855} C_VEL
LIN {X 0,Y 509.278,Z 552.387,A -85,B 0,C 180,E1 -5486.045,E2 -5486.045} C_VEL
LIN {X 0,Y 509.201,Z 554.282,A -85,B 0,C 180,E1 -5486.837,E2 -5486.837} C_VEL
LIN {X 0,Y 509.189,Z 555.705,A -85,B 0,C 180,E1 -5487.628,E2 -5487.628} C_VEL
LIN {X 0,Y 509.081,Z 557.34,A -85,B 0,C 180,E1 -5489.21,E2 -5489.21} C_VEL
LIN {X 0,Y 509.082,Z 557.567,A -85,B 0,C 180,E1 -5490.001,E2 -5490.001} C_VEL
LIN {X 0,Y 509.112,Z 556.745,A -85,B 0,C 180,E1 -5491.583,E2 -5491.583} C_VEL
LIN {X 0,Y 509.19,Z 555.747,A -85,B 0,C 180,E1 -5492.374,E2 -5492.374} C_VEL
LIN {X 0,Y 509.202,Z 554.336,A -85,B 0,C 180,E1 -5493.166,E2 -5493.166} C_VEL
LIN {X 0,Y 509.207,Z 551.369,A -85,B 0,C 180,E1 -5494.354,E2 -5494.354} C_VEL
LIN {X 0,Y 509.309,Z 547.353,A -85,B 0,C 180,E1 -5495.544,E2 -5495.544} C_VEL
LIN {X 0,Y 509.374,Z 541.617,A -85,B 0,C 180,E1 -5496.845,E2 -5496.845} C_VEL
LIN {X 0,Y 509.509,Z 534.399,A -85,B 0,C 180,E1 -5498.128,E2 -5498.128} C_VEL
LIN {X 0,Y 509.721,Z 526.01,A -85,B 0,C 180,E1 -5499.324,E2 -5499.324} C_VEL
LIN {X 0,Y 509.973,Z 517.382,A -85,B 0,C 180,E1 -5500.321,E2 -5500.321} C_VEL
LIN {X 0,Y 510.342,Z 506.743,A -85,B 0,C 180,E1 -5501.317,E2 -5501.317} C_VEL
LIN {X 0,Y 510.64,Z 495.431,A -85,B 0,C 180,E1 -5502.17,E2 -5502.17} C_VEL
LIN {X 0,Y 510.935,Z 484.575,A -85,B 0,C 180,E1 -5502.815,E2 -5502.815} C_VEL
LIN {X 0,Y 511.212,Z 472.512,A -85,B 0,C 180,E1 -5503.364,E2 -5503.364} C_VEL
LIN {X 0,Y 511.473,Z 459.487,A -85,B 0,C 180,E1 -5503.787,E2 -5503.787} C_VEL
LIN {X 0,Y 511.687,Z 445.555,A -85,B 0,C 180,E1 -5504.06,E2 -5504.06} C_VEL
LIN {X 0,Y 512.054,Z 356.55,A -85,B 0,C 180,E1 -5505.344,E2 -5505.344} C_VEL
LIN {X 0,Y 510.305,Z 344.22,A -85,B 0,C 180,E1 -5505.598,E2 -5505.598} C_VEL
LIN {X 0,Y 510.775,Z 323.704,A -85,B 0,C 180,E1 -5508.657,E2 -5508.657} C_VEL
LIN {X 0,Y 511.365,Z 304.372,A -85,B 0,C 180,E1 -5511.569,E2 -5511.569} C_VEL
LIN {X 0,Y 511.823,Z 287.799,A -85,B 0,C 180,E1 -5514.11,E2 -5514.11} C_VEL
LIN {X 0,Y 510.075,Z 278.046,A -85,B 0,C 180,E1 -5515.721,E2 -5515.721} C_VEL
LIN {X 0,Y 509.846,Z 276.978,A -85,B 0,C 180,E1 -5515.926,E2 -5515.926} C_VEL
LIN {X 0,Y 509.844,Z 276.978,A -85,B 0,C 180,E1 -5518.844,E2 -5518.844} C_VEL
LIN {X 0,Y 509.811,Z 276.977,A -85,B 0,C 180,E1 -5521.589,E2 -5521.589} C_VEL
LIN {X 0,Y 509.825,Z 276.981,A -85,B 0,C 180,E1 -5524.413,E2 -5524.413} C_VEL
LIN {X 0,Y 509.782,Z 276.98,A -85,B 0,C 180,E1 -5527.341,E2 -5527.341} C_VEL
LIN {X 0,Y 509.8,Z 276.982,A -85,B 0,C 180,E1 -5530.383,E2 -5530.383} C_VEL
LIN {X 0,Y 509.78,Z 276.983,A -85,B 0,C 180,E1 -5533.056,E2 -5533.056} C_VEL
LIN {X 0,Y 509.804,Z 276.977,A -85,B 0,C 180,E1 -5535.791,E2 -5535.791} C_VEL
LIN {X 0,Y 509.811,Z 276.983,A -85,B 0,C 180,E1 -5538.57,E2 -5538.57} C_VEL
LIN {X 0,Y 509.8,Z 276.978,A -85,B 0,C 180,E1 -5541.789,E2 -5541.789} C_VEL
LIN {X 0,Y 509.8,Z 276.984,A -85,B 0,C 180,E1 -5544.619,E2 -5544.619} C_VEL
LIN {X 0,Y 509.832,Z 276.974,A -85,B 0,C 180,E1 -5547.478,E2 -5547.478} C_VEL
LIN {X 0,Y 509.83,Z 276.977,A -85,B 0,C 180,E1 -5550.272,E2 -5550.272} C_VEL
LIN {X 0,Y 509.84,Z 276.979,A -85,B 0,C 180,E1 -5552.941,E2 -5552.941} C_VEL
LIN {X 0,Y 509.784,Z 276.984,A -85,B 0,C 180,E1 -5556.434,E2 -5556.434} C_VEL
LIN {X 0,Y 509.872,Z 276.969,A -85,B 0,C 180,E1 -5559.842,E2 -5559.842} C_VEL
LIN {X 0,Y 509.831,Z 276.978,A -85,B 0,C 180,E1 -5563.173,E2 -5563.173} C_VEL
LIN {X 0,Y 509.82,Z 276.976,A -85,B 0,C 180,E1 -5565.632,E2 -5565.632} C_VEL
LIN {X 0,Y 509.892,Z 276.974,A -85,B 0,C 180,E1 -5568.874,E2 -5568.874} C_VEL
LIN {X 0,Y 509.912,Z 276.965,A -85,B 0,C 180,E1 -5572.077,E2 -5572.077} C_VEL
LIN {X 0,Y 509.94,Z 276.965,A -85,B 0,C 180,E1 -5574.463,E2 -5574.463} C_VEL
LIN {X 0,Y 510.011,Z 276.952,A -85,B 0,C 180,E1 -5577.63,E2 -5577.63} C_VEL
LIN {X 0,Y 510.01,Z 276.953,A -85,B 0,C 180,E1 -5580,E2 -5580} C_VEL
LIN {X 0,Y 510.013,Z 276.955,A -85,B 0,C 180,E1 -5582.369,E2 -5582.369} C_VEL
LIN {X 0,Y 509.942,Z 276.962,A -85,B 0,C 180,E1 -5585.536,E2 -5585.536} C_VEL
LIN {X 0,Y 509.913,Z 276.965,A -85,B 0,C 180,E1 -5587.922,E2 -5587.922} C_VEL
LIN {X 0,Y 509.897,Z 276.972,A -85,B 0,C 180,E1 -5591.125,E2 -5591.125} C_VEL
LIN {X 0,Y 509.826,Z 276.978,A -85,B 0,C 180,E1 -5594.367,E2 -5594.367} C_VEL
LIN {X 0,Y 509.865,Z 276.971,A -85,B 0,C 180,E1 -5597.652,E2 -5597.652} C_VEL
LIN {X 0,Y 509.851,Z 276.975,A -85,B 0,C 180,E1 -5600.402,E2 -5600.402} C_VEL
LIN {X 0,Y 509.802,Z 276.979,A -85,B 0,C 180,E1 -5603.564,E2 -5603.564} C_VEL
LIN {X 0,Y 509.881,Z 276.971,A -85,B 0,C 180,E1 -5606.38,E2 -5606.38} C_VEL
LIN {X 0,Y 509.854,Z 276.977,A -85,B 0,C 180,E1 -5608.845,E2 -5608.845} C_VEL
LIN {X 0,Y 509.796,Z 276.98,A -85,B 0,C 180,E1 -5611.591,E2 -5611.591} C_VEL
LIN {X 0,Y 509.827,Z 276.978,A -85,B 0,C 180,E1 -5614.415,E2 -5614.415} C_VEL
LIN {X 0,Y 509.793,Z 276.983,A -85,B 0,C 180,E1 -5617.342,E2 -5617.342} C_VEL
LIN {X 0,Y 509.838,Z 276.976,A -85,B 0,C 180,E1 -5620.382,E2 -5620.382} C_VEL
LIN {X 0,Y 509.802,Z 276.984,A -85,B 0,C 180,E1 -5623.064,E2 -5623.064} C_VEL
LIN {X 0,Y 509.811,Z 276.978,A -85,B 0,C 180,E1 -5625.794,E2 -5625.794} C_VEL
LIN {X 0,Y 509.849,Z 276.976,A -85,B 0,C 180,E1 -5628.577,E2 -5628.577} C_VEL
LIN {X 0,Y 509.842,Z 276.974,A -85,B 0,C 180,E1 -5631.787,E2 -5631.787} C_VEL
LIN {X 0,Y 509.818,Z 276.977,A -85,B 0,C 180,E1 -5633.764,E2 -5633.764} C_VEL
LIN {X 0,Y 509.153,Z 277.062,A -85,B 0,C 180,E1 -5634.424,E2 -5634.424} C_VEL
LIN {X 0,Y 506.335,Z 277.415,A -85,B 0,C 180,E1 -5635.496,E2 -5635.496} C_VEL
LIN {X 0,Y 503.941,Z 277.715,A -85,B 0,C 180,E1 -5636.359,E2 -5636.359} C_VEL
LIN {X 0,Y 502.891,Z 277.844,A -85,B 0,C 180,E1 -5637.025,E2 -5637.025} C_VEL
LIN {X 0,Y 502.794,Z 277.854,A -85,B 0,C 180,E1 -5637.251,E2 -5637.251} C_VEL
LIN {X 0,Y 502.805,Z 277.85,A -85,B 0,C 180,E1 -5640.066,E2 -5640.066} C_VEL
LIN {X 0,Y 502.826,Z 277.85,A -85,B 0,C 180,E1 -5642.534,E2 -5642.534} C_VEL
LIN {X 0,Y 502.819,Z 277.853,A -85,B 0,C 180,E1 -5645.3,E2 -5645.3} C_VEL
LIN {X 0,Y 502.774,Z 277.854,A -85,B 0,C 180,E1 -5647.827,E2 -5647.827} C_VEL
LIN {X 0,Y 502.82,Z 277.849,A -85,B 0,C 180,E1 -5650.401,E2 -5650.401} C_VEL
LIN {X 0,Y 502.83,Z 277.853,A -85,B 0,C 180,E1 -5652.932,E2 -5652.932} C_VEL
LIN {X 0,Y 502.841,Z 277.849,A -85,B 0,C 180,E1 -5655.429,E2 -5655.429} C_VEL
LIN {X 0,Y 502.874,Z 277.845,A -85,B 0,C 180,E1 -5658.717,E2 -5658.717} C_VEL
LIN {X 0,Y 502.9,Z 277.838,A -85,B 0,C 180,E1 -5661.966,E2 -5661.966} C_VEL
LIN {X 0,Y 502.935,Z 277.834,A -85,B 0,C 180,E1 -5664.386,E2 -5664.386} C_VEL
LIN {X 0,Y 503.023,Z 277.825,A -85,B 0,C 180,E1 -5667.597,E2 -5667.597} C_VEL
LIN {X 0,Y 503.025,Z 277.822,A -85,B 0,C 180,E1 -5669.999,E2 -5669.999} C_VEL
LIN {X 0,Y 503.023,Z 277.823,A -85,B 0,C 180,E1 -5672.401,E2 -5672.401} C_VEL
LIN {X 0,Y 502.93,Z 277.836,A -85,B 0,C 180,E1 -5675.612,E2 -5675.612} C_VEL
LIN {X 0,Y 502.897,Z 277.838,A -85,B 0,C 180,E1 -5678.031,E2 -5678.031} C_VEL
LIN {X 0,Y 502.886,Z 277.844,A -85,B 0,C 180,E1 -5681.281,E2 -5681.281} C_VEL
LIN {X 0,Y 502.837,Z 277.847,A -85,B 0,C 180,E1 -5684.568,E2 -5684.568} C_VEL
LIN {X 0,Y 502.852,Z 277.844,A -85,B 0,C 180,E1 -5687.904,E2 -5687.904} C_VEL
LIN {X 0,Y 502.818,Z 277.849,A -85,B 0,C 180,E1 -5690.534,E2 -5690.534} C_VEL
LIN {X 0,Y 502.792,Z 277.858,A -85,B 0,C 180,E1 -5693.037,E2 -5693.037} C_VEL
LIN {X 0,Y 502.826,Z 277.849,A -85,B 0,C 180,E1 -5695.672,E2 -5695.672} C_VEL
LIN {X 0,Y 502.824,Z 277.847,A -85,B 0,C 180,E1 -5698.369,E2 -5698.369} C_VEL
LIN {X 0,Y 502.776,Z 277.856,A -85,B 0,C 180,E1 -5701.496,E2 -5701.496} C_VEL
LIN {X 0,Y 502.783,Z 277.852,A -85,B 0,C 180,E1 -5704.441,E2 -5704.441} C_VEL
LIN {X 0,Y 502.757,Z 277.863,A -85,B 0,C 180,E1 -5707.175,E2 -5707.175} C_VEL
LIN {X 0,Y 502.805,Z 277.851,A -85,B 0,C 180,E1 -5710.007,E2 -5710.007} C_VEL
LIN {X 0,Y 502.9,Z 277.903,A -85,B 0,C 180,E1 -5713.595,E2 -5713.595} C_VEL
LIN {X 0,Y 503.374,Z 282.717,A -85,B 0,C 180,E1 -5714.599,E2 -5714.599} C_VEL
LIN {X 0,Y 503.232,Z 291.238,A -85,B 0,C 180,E1 -5716.273,E2 -5716.273} C_VEL
LIN {X 0,Y 505.427,Z 302.168,A -85,B 0,C 180,E1 -5716.51,E2 -5716.51} C_VEL
LIN {X 0,Y 504.783,Z 397.622,A -85,B 0,C 180,E1 -5717.934,E2 -5717.934} C_VEL
LIN {X 0,Y 504.627,Z 410.861,A -85,B 0,C 180,E1 -5718.293,E2 -5718.293} C_VEL
LIN {X 0,Y 504.35,Z 423.492,A -85,B 0,C 180,E1 -5718.797,E2 -5718.797} C_VEL
LIN {X 0,Y 504.046,Z 435.503,A -85,B 0,C 180,E1 -5719.451,E2 -5719.451} C_VEL
LIN {X 0,Y 503.672,Z 447.039,A -85,B 0,C 180,E1 -5720.264,E2 -5720.264} C_VEL
LIN {X 0,Y 503.332,Z 457.477,A -85,B 0,C 180,E1 -5721.184,E2 -5721.184} C_VEL
LIN {X 0,Y 503.023,Z 467.318,A -85,B 0,C 180,E1 -5722.27,E2 -5722.27} C_VEL
LIN {X 0,Y 502.801,Z 474.994,A -85,B 0,C 180,E1 -5723.306,E2 -5723.306} C_VEL
LIN {X 0,Y 502.516,Z 482.768,A -85,B 0,C 180,E1 -5724.596,E2 -5724.596} C_VEL
LIN {X 0,Y 502.356,Z 489.215,A -85,B 0,C 180,E1 -5725.972,E2 -5725.972} C_VEL
LIN {X 0,Y 502.249,Z 494.523,A -85,B 0,C 180,E1 -5727.48,E2 -5727.48} C_VEL
LIN {X 0,Y 502.116,Z 497.858,A -85,B 0,C 180,E1 -5728.81,E2 -5728.81} C_VEL
LIN {X 0,Y 502.049,Z 500.07,A -85,B 0,C 180,E1 -5730.205,E2 -5730.205} C_VEL
LIN {X 0,Y 502.025,Z 501.116,A -85,B 0,C 180,E1 -5731.866,E2 -5731.866} C_VEL
LIN {X 0,Y 502.042,Z 500.605,A -85,B 0,C 180,E1 -5733.387,E2 -5733.387} C_VEL
LIN {X 0,Y 502.062,Z 499.604,A -85,B 0,C 180,E1 -5734.282,E2 -5734.282} C_VEL
LIN {X 0,Y 502.122,Z 497.543,A -85,B 0,C 180,E1 -5735.459,E2 -5735.459} C_VEL
LIN {X 0,Y 502.303,Z 493.638,A -85,B 0,C 180,E1 -5736.936,E2 -5736.936} C_VEL
LIN {X 0,Y 502.373,Z 488.881,A -85,B 0,C 180,E1 -5738.24,E2 -5738.24} C_VEL
LIN {X 0,Y 502.531,Z 482.714,A -85,B 0,C 180,E1 -5739.536,E2 -5739.536} C_VEL
LIN {X 0,Y 502.788,Z 474.941,A -85,B 0,C 180,E1 -5740.824,E2 -5740.824} C_VEL
LIN {X 0,Y 503.061,Z 466.92,A -85,B 0,C 180,E1 -5741.898,E2 -5741.898} C_VEL
LIN {X 0,Y 503.406,Z 457.208,A -85,B 0,C 180,E1 -5742.952,E2 -5742.952} C_VEL
LIN {X 0,Y 503.719,Z 447.625,A -85,B 0,C 180,E1 -5743.797,E2 -5743.797} C_VEL
LIN {X 0,Y 504.052,Z 435.743,A -85,B 0,C 180,E1 -5744.638,E2 -5744.638} C_VEL
LIN {X 0,Y 504.339,Z 424.267,A -85,B 0,C 180,E1 -5745.267,E2 -5745.267} C_VEL
LIN {X 0,Y 504.523,Z 411.378,A -85,B 0,C 180,E1 -5745.788,E2 -5745.788} C_VEL
LIN {X 0,Y 504.751,Z 398.297,A -85,B 0,C 180,E1 -5746.142,E2 -5746.142} C_VEL
LIN {X 0,Y 505.327,Z 301.602,A -85,B 0,C 180,E1 -5747.602,E2 -5747.602} C_VEL
LIN {X 0,Y 503.171,Z 290.415,A -85,B 0,C 180,E1 -5747.849,E2 -5747.849} C_VEL
LIN {X 0,Y 502.932,Z 278.494,A -85,B 0,C 180,E1 -5749.737,E2 -5749.737} C_VEL
LIN {X 0,Y 502.818,Z 277.853,A -85,B 0,C 180,E1 -5749.887,E2 -5749.887} C_VEL
LIN {X 0,Y 502.877,Z 277.848,A -85,B 0,C 180,E1 -5752.813,E2 -5752.813} C_VEL
LIN {X 0,Y 502.815,Z 277.856,A -85,B 0,C 180,E1 -5755.19,E2 -5755.19} C_VEL
LIN {X 0,Y 502.965,Z 277.833,A -85,B 0,C 180,E1 -5757.598,E2 -5757.598} C_VEL
LIN {X 0,Y 502.961,Z 277.83,A -85,B 0,C 180,E1 -5760,E2 -5760} C_VEL
LIN {X 0,Y 502.966,Z 277.832,A -85,B 0,C 180,E1 -5762.403,E2 -5762.403} C_VEL
LIN {X 0,Y 502.889,Z 277.84,A -85,B 0,C 180,E1 -5765.614,E2 -5765.614} C_VEL
LIN {X 0,Y 502.843,Z 277.844,A -85,B 0,C 180,E1 -5768.035,E2 -5768.035} C_VEL
LIN {X 0,Y 502.844,Z 277.849,A -85,B 0,C 180,E1 -5771.284,E2 -5771.284} C_VEL
LIN {X 0,Y 502.801,Z 277.853,A -85,B 0,C 180,E1 -5774.573,E2 -5774.573} C_VEL
LIN {X 0,Y 502.807,Z 277.847,A -85,B 0,C 180,E1 -5777.909,E2 -5777.909} C_VEL
LIN {X 0,Y 502.776,Z 277.853,A -85,B 0,C 180,E1 -5780.539,E2 -5780.539} C_VEL
LIN {X 0,Y 502.742,Z 277.862,A -85,B 0,C 180,E1 -5783.043,E2 -5783.043} C_VEL
LIN {X 0,Y 502.792,Z 277.85,A -85,B 0,C 180,E1 -5785.679,E2 -5785.679} C_VEL
LIN {X 0,Y 502.793,Z 277.851,A -85,B 0,C 180,E1 -5788.376,E2 -5788.376} C_VEL
LIN {X 0,Y 502.751,Z 277.859,A -85,B 0,C 180,E1 -5791.503,E2 -5791.503} C_VEL
LIN {X 0,Y 502.764,Z 277.853,A -85,B 0,C 180,E1 -5794.448,E2 -5794.448} C_VEL
LIN {X 0,Y 502.741,Z 277.863,A -85,B 0,C 180,E1 -5797.182,E2 -5797.182} C_VEL
LIN {X 0,Y 502.791,Z 277.851,A -85,B 0,C 180,E1 -5800.015,E2 -5800.015} C_VEL
LIN {X 0,Y 502.769,Z 277.852,A -85,B 0,C 180,E1 -5802.203,E2 -5802.203} C_VEL
LIN {X 0,Y 502.77,Z 277.86,A -85,B 0,C 180,E1 -5805.472,E2 -5805.472} C_VEL
LIN {X 0,Y 502.794,Z 277.855,A -85,B 0,C 180,E1 -5808.938,E2 -5808.938} C_VEL
LIN {X 0,Y 502.768,Z 277.855,A -85,B 0,C 180,E1 -5812.05,E2 -5812.05} C_VEL
LIN {X 0,Y 502.777,Z 277.859,A -85,B 0,C 180,E1 -5815.038,E2 -5815.038} C_VEL
LIN {X 0,Y 502.765,Z 277.861,A -85,B 0,C 180,E1 -5817.919,E2 -5817.919} C_VEL
LIN {X 0,Y 502.799,Z 277.855,A -85,B 0,C 180,E1 -5820.715,E2 -5820.715} C_VEL
LIN {X 0,Y 502.832,Z 277.855,A -85,B 0,C 180,E1 -5823.447,E2 -5823.447} C_VEL
LIN {X 0,Y 502.905,Z 278.031,A -85,B 0,C 180,E1 -5824.609,E2 -5824.609} C_VEL
LIN {X 0,Y 504.3,Z 286.635,A -85,B 0,C 180,E1 -5825.948,E2 -5825.948} C_VEL
LIN {X 0,Y 504.003,Z 305.683,A -85,B 0,C 180,E1 -5828.747,E2 -5828.747} C_VEL
LIN {X 0,Y 503.556,Z 327.193,A -85,B 0,C 180,E1 -5831.881,E2 -5831.881} C_VEL
LIN {X 0,Y 503.217,Z 343.015,A -85,B 0,C 180,E1 -5834.183,E2 -5834.183} C_VEL
LIN {X 0,Y 505.283,Z 358.101,A -85,B 0,C 180,E1 -5834.483,E2 -5834.483} C_VEL
LIN {X 0,Y 504.652,Z 452.566,A -85,B 0,C 180,E1 -5835.897,E2 -5835.897} C_VEL
LIN {X 0,Y 504.37,Z 465.699,A -85,B 0,C 180,E1 -5836.249,E2 -5836.249} C_VEL
LIN {X 0,Y 504.06,Z 478.421,A -85,B 0,C 180,E1 -5836.754,E2 -5836.754} C_VEL
LIN {X 0,Y 503.78,Z 490.035,A -85,B 0,C 180,E1 -5837.379,E2 -5837.379} C_VEL
LIN {X 0,Y 503.368,Z 502.156,A -85,B 0,C 180,E1 -5838.22,E2 -5838.22} C_VEL
LIN {X 0,Y 503.1,Z 512.626,A -85,B 0,C 180,E1 -5839.132,E2 -5839.132} C_VEL
LIN {X 0,Y 502.757,Z 522.016,A -85,B 0,C 180,E1 -5840.142,E2 -5840.142} C_VEL
LIN {X 0,Y 502.497,Z 531.141,A -85,B 0,C 180,E1 -5841.355,E2 -5841.355} C_VEL
LIN {X 0,Y 502.332,Z 538.494,A -85,B 0,C 180,E1 -5842.566,E2 -5842.566} C_VEL
LIN {X 0,Y 502.234,Z 543.455,A -85,B 0,C 180,E1 -5843.574,E2 -5843.574} C_VEL
LIN {X 0,Y 502.179,Z 548.279,A -85,B 0,C 180,E1 -5844.783,E2 -5844.783} C_VEL
LIN {X 0,Y 502.171,Z 551.968,A -85,B 0,C 180,E1 -5845.989,E2 -5845.989} C_VEL
LIN {X 0,Y 502.123,Z 553.872,A -85,B 0,C 180,E1 -5846.792,E2 -5846.792} C_VEL
LIN {X 0,Y 502.12,Z 555.3,A -85,B 0,C 180,E1 -5847.595,E2 -5847.595} C_VEL
LIN {X 0,Y 501.997,Z 556.944,A -85,B 0,C 180,E1 -5849.199,E2 -5849.199} C_VEL
LIN {X 0,Y 501.995,Z 557.172,A -85,B 0,C 180,E1 -5850.001,E2 -5850.001} C_VEL
LIN {X 0,Y 502.036,Z 556.352,A -85,B 0,C 180,E1 -5851.605,E2 -5851.605} C_VEL
LIN {X 0,Y 502.121,Z 555.354,A -85,B 0,C 180,E1 -5852.408,E2 -5852.408} C_VEL
LIN {X 0,Y 502.123,Z 553.94,A -85,B 0,C 180,E1 -5853.21,E2 -5853.21} C_VEL
LIN {X 0,Y 502.105,Z 550.968,A -85,B 0,C 180,E1 -5854.416,E2 -5854.416} C_VEL
LIN {X 0,Y 502.221,Z 546.946,A -85,B 0,C 180,E1 -5855.622,E2 -5855.622} C_VEL
LIN {X 0,Y 502.325,Z 540.846,A -85,B 0,C 180,E1 -5857.012,E2 -5857.012} C_VEL
LIN {X 0,Y 502.46,Z 533.97,A -85,B 0,C 180,E1 -5858.243,E2 -5858.243} C_VEL
LIN {X 0,Y 502.674,Z 525.566,A -85,B 0,C 180,E1 -5859.456,E2 -5859.456} C_VEL
LIN {X 0,Y 502.96,Z 516.918,A -85,B 0,C 180,E1 -5860.466,E2 -5860.466} C_VEL
LIN {X 0,Y 503.335,Z 506.258,A -85,B 0,C 180,E1 -5861.477,E2 -5861.477} C_VEL
LIN {X 0,Y 503.641,Z 494.608,A -85,B 0,C 180,E1 -5862.363,E2 -5862.363} C_VEL
LIN {X 0,Y 503.975,Z 484.015,A -85,B 0,C 180,E1 -5862.995,E2 -5862.995} C_VEL
LIN {X 0,Y 504.29,Z 471.904,A -85,B 0,C 180,E1 -5863.551,E2 -5863.551} C_VEL
LIN {X 0,Y 504.577,Z 458.795,A -85,B 0,C 180,E1 -5863.979,E2 -5863.979} C_VEL
LIN {X 0,Y 504.773,Z 446.325,A -85,B 0,C 180,E1 -5864.231,E2 -5864.231} C_VEL
LIN {X 0,Y 505.168,Z 357.176,A -85,B 0,C 180,E1 -5865.544,E2 -5865.544} C_VEL
LIN {X 0,Y 503.268,Z 343.833,A -85,B 0,C 180,E1 -5865.826,E2 -5865.826} C_VEL
LIN {X 0,Y 503.781,Z 324.721,A -85,B 0,C 180,E1 -5868.714,E2 -5868.714} C_VEL
LIN {X 0,Y 504.395,Z 305.42,A -85,B 0,C 180,E1 -5871.668,E2 -5871.668} C_VEL
LIN {X 0,Y 504.894,Z 288.868,A -85,B 0,C 180,E1 -5874.243,E2 -5874.243} C_VEL
LIN {X 0,Y 502.797,Z 277.857,A -85,B 0,C 180,E1 -5876.122,E2 -5876.122} C_VEL
LIN {X 0,Y 502.807,Z 277.85,A -85,B 0,C 180,E1 -5879.287,E2 -5879.287} C_VEL
LIN {X 0,Y 502.775,Z 277.855,A -85,B 0,C 180,E1 -5882.083,E2 -5882.083} C_VEL
LIN {X 0,Y 502.781,Z 277.856,A -85,B 0,C 180,E1 -5884.965,E2 -5884.965} C_VEL
LIN {X 0,Y 502.752,Z 277.861,A -85,B 0,C 180,E1 -5888.479,E2 -5888.479} C_VEL
LIN {X 0,Y 502.758,Z 277.858,A -85,B 0,C 180,E1 -5891.069,E2 -5891.069} C_VEL
LIN {X 0,Y 502.769,Z 277.859,A -85,B 0,C 180,E1 -5894.528,E2 -5894.528} C_VEL
LIN {X 0,Y 502.747,Z 277.857,A -85,B 0,C 180,E1 -5897.855,E2 -5897.855} C_VEL
LIN {X 0,Y 502.765,Z 277.858,A -85,B 0,C 180,E1 -5901.02,E2 -5901.02} C_VEL
LIN {X 0,Y 502.746,Z 277.859,A -85,B 0,C 180,E1 -5904.168,E2 -5904.168} C_VEL
LIN {X 0,Y 502.778,Z 277.857,A -85,B 0,C 180,E1 -5906.997,E2 -5906.997} C_VEL
LIN {X 0,Y 502.786,Z 277.853,A -85,B 0,C 180,E1 -5910.063,E2 -5910.063} C_VEL
LIN {X 0,Y 502.791,Z 277.856,A -85,B 0,C 180,E1 -5912.53,E2 -5912.53} C_VEL
LIN {X 0,Y 502.739,Z 277.859,A -85,B 0,C 180,E1 -5915.312,E2 -5915.312} C_VEL
LIN {X 0,Y 502.745,Z 277.857,A -85,B 0,C 180,E1 -5917.824,E2 -5917.824} C_VEL
LIN {X 0,Y 502.779,Z 277.857,A -85,B 0,C 180,E1 -5920.398,E2 -5920.398} C_VEL
LIN {X 0,Y 502.776,Z 277.86,A -85,B 0,C 180,E1 -5922.929,E2 -5922.929} C_VEL
LIN {X 0,Y 502.799,Z 277.852,A -85,B 0,C 180,E1 -5925.427,E2 -5925.427} C_VEL
LIN {X 0,Y 502.861,Z 277.848,A -85,B 0,C 180,E1 -5928.716,E2 -5928.716} C_VEL
LIN {X 0,Y 502.863,Z 277.843,A -85,B 0,C 180,E1 -5931.966,E2 -5931.966} C_VEL
LIN {X 0,Y 502.894,Z 277.842,A -85,B 0,C 180,E1 -5934.386,E2 -5934.386} C_VEL
LIN {X 0,Y 502.982,Z 277.828,A -85,B 0,C 180,E1 -5937.597,E2 -5937.597} C_VEL
LIN {X 0,Y 502.982,Z 277.828,A -85,B 0,C 180,E1 -5940,E2 -5940} C_VEL
LIN {X 0,Y 502.983,Z 277.831,A -85,B 0,C 180,E1 -5942.402,E2 -5942.402} C_VEL
LIN {X 0,Y 502.895,Z 277.839,A -85,B 0,C 180,E1 -5945.614,E2 -5945.614} C_VEL
LIN {X 0,Y 502.864,Z 277.843,A -85,B 0,C 180,E1 -5948.034,E2 -5948.034} C_VEL
LIN {X 0,Y 502.864,Z 277.846,A -85,B 0,C 180,E1 -5951.283,E2 -5951.283} C_VEL
LIN {X 0,Y 502.807,Z 277.855,A -85,B 0,C 180,E1 -5954.572,E2 -5954.572} C_VEL
LIN {X 0,Y 502.825,Z 277.848,A -85,B 0,C 180,E1 -5957.908,E2 -5957.908} C_VEL
LIN {X 0,Y 502.794,Z 277.856,A -85,B 0,C 180,E1 -5960.537,E2 -5960.537} C_VEL
LIN {X 0,Y 502.76,Z 277.861,A -85,B 0,C 180,E1 -5963.042,E2 -5963.042} C_VEL
LIN {X 0,Y 502.808,Z 277.85,A -85,B 0,C 180,E1 -5965.677,E2 -5965.677} C_VEL
LIN {X 0,Y 502.812,Z 277.852,A -85,B 0,C 180,E1 -5968.374,E2 -5968.374} C_VEL
LIN {X 0,Y 502.767,Z 277.857,A -85,B 0,C 180,E1 -5971.501,E2 -5971.501} C_VEL
LIN {X 0,Y 502.78,Z 277.856,A -85,B 0,C 180,E1 -5974.446,E2 -5974.446} C_VEL
LIN {X 0,Y 502.756,Z 277.862,A -85,B 0,C 180,E1 -5977.18,E2 -5977.18} C_VEL
LIN {X 0,Y 502.803,Z 277.851,A -85,B 0,C 180,E1 -5980.013,E2 -5980.013} C_VEL
LIN {X 0,Y 502.752,Z 277.862,A -85,B 0,C 180,E1 -5983.233,E2 -5983.233} C_VEL
LIN {X 0,Y 502.77,Z 277.855,A -85,B 0,C 180,E1 -5985.663,E2 -5985.663} C_VEL
LIN {X 0,Y 502.812,Z 277.849,A -85,B 0,C 180,E1 -5987.866,E2 -5987.866} C_VEL
LIN {X 0,Y 502.806,Z 277.855,A -85,B 0,C 180,E1 -5991.027,E2 -5991.027} C_VEL
LIN {X 0,Y 502.772,Z 277.855,A -85,B 0,C 180,E1 -5994.169,E2 -5994.169} C_VEL
LIN {X 0,Y 502.794,Z 277.854,A -85,B 0,C 180,E1 -5997.251,E2 -5997.251} C_VEL
LIN {X 0,Y 502.093,Z 277.94,A -85,B 0,C 180,E1 -5997.92,E2 -5997.92} C_VEL
LIN {X 0,Y 499.229,Z 278.301,A -85,B 0,C 180,E1 -5999.005,E2 -5999.005} C_VEL
LIN {X 0,Y 496.836,Z 278.596,A -85,B 0,C 180,E1 -5999.88,E2 -5999.88} C_VEL
LIN {X 0,Y 495.821,Z 278.723,A -85,B 0,C 180,E1 -6000.556,E2 -6000.556} C_VEL
LIN {X 0,Y 495.744,Z 278.731,A -85,B 0,C 180,E1 -6000.785,E2 -6000.785} C_VEL
LIN {X 0,Y 495.783,Z 278.725,A -85,B 0,C 180,E1 -6003.933,E2 -6003.933} C_VEL
LIN {X 0,Y 495.753,Z 278.733,A -85,B 0,C 180,E1 -6007.14,E2 -6007.14} C_VEL
LIN {X 0,Y 495.767,Z 278.727,A -85,B 0,C 180,E1 -6010.11,E2 -6010.11} C_VEL
LIN {X 0,Y 495.783,Z 278.729,A -85,B 0,C 180,E1 -6012.682,E2 -6012.682} C_VEL
LIN {X 0,Y 495.786,Z 278.729,A -85,B 0,C 180,E1 -6015.217,E2 -6015.217} C_VEL
LIN {X 0,Y 495.849,Z 278.719,A -85,B 0,C 180,E1 -6018.555,E2 -6018.555} C_VEL
LIN {X 0,Y 495.871,Z 278.714,A -85,B 0,C 180,E1 -6021.852,E2 -6021.852} C_VEL
LIN {X 0,Y 495.893,Z 278.711,A -85,B 0,C 180,E1 -6024.306,E2 -6024.306} C_VEL
LIN {X 0,Y 495.991,Z 278.701,A -85,B 0,C 180,E1 -6027.563,E2 -6027.563} C_VEL
LIN {X 0,Y 495.996,Z 278.698,A -85,B 0,C 180,E1 -6029.999,E2 -6029.999} C_VEL
LIN {X 0,Y 495.991,Z 278.7,A -85,B 0,C 180,E1 -6032.435,E2 -6032.435} C_VEL
LIN {X 0,Y 495.886,Z 278.713,A -85,B 0,C 180,E1 -6035.692,E2 -6035.692} C_VEL
LIN {X 0,Y 495.868,Z 278.714,A -85,B 0,C 180,E1 -6038.146,E2 -6038.146} C_VEL
LIN {X 0,Y 495.867,Z 278.717,A -85,B 0,C 180,E1 -6041.442,E2 -6041.442} C_VEL
LIN {X 0,Y 495.782,Z 278.728,A -85,B 0,C 180,E1 -6044.78,E2 -6044.78} C_VEL
LIN {X 0,Y 495.779,Z 278.729,A -85,B 0,C 180,E1 -6047.316,E2 -6047.316} C_VEL
LIN {X 0,Y 495.767,Z 278.727,A -85,B 0,C 180,E1 -6049.887,E2 -6049.887} C_VEL
LIN {X 0,Y 495.751,Z 278.732,A -85,B 0,C 180,E1 -6052.859,E2 -6052.859} C_VEL
LIN {X 0,Y 495.783,Z 278.724,A -85,B 0,C 180,E1 -6056.064,E2 -6056.064} C_VEL
LIN {X 0,Y 495.761,Z 278.73,A -85,B 0,C 180,E1 -6058.811,E2 -6058.811} C_VEL
LIN {X 0,Y 495.738,Z 278.731,A -85,B 0,C 180,E1 -6061.723,E2 -6061.723} C_VEL
LIN {X 0,Y 495.752,Z 278.729,A -85,B 0,C 180,E1 -6064.692,E2 -6064.692} C_VEL
LIN {X 0,Y 495.708,Z 278.737,A -85,B 0,C 180,E1 -6067.557,E2 -6067.557} C_VEL
LIN {X 0,Y 495.771,Z 278.727,A -85,B 0,C 180,E1 -6070.049,E2 -6070.049} C_VEL
LIN {X 0,Y 495.863,Z 278.846,A -85,B 0,C 180,E1 -6073.478,E2 -6073.478} C_VEL
LIN {X 0,Y 496.401,Z 283.303,A -85,B 0,C 180,E1 -6074.416,E2 -6074.416} C_VEL
LIN {X 0,Y 496.239,Z 291.292,A -85,B 0,C 180,E1 -6076.043,E2 -6076.043} C_VEL
LIN {X 0,Y 498.608,Z 303.946,A -85,B 0,C 180,E1 -6076.318,E2 -6076.318} C_VEL
LIN {X 0,Y 497.902,Z 398.585,A -85,B 0,C 180,E1 -6077.761,E2 -6077.761} C_VEL
LIN {X 0,Y 497.745,Z 411.969,A -85,B 0,C 180,E1 -6078.136,E2 -6078.136} C_VEL
LIN {X 0,Y 497.43,Z 424.71,A -85,B 0,C 180,E1 -6078.662,E2 -6078.662} C_VEL
LIN {X 0,Y 497.1,Z 436.106,A -85,B 0,C 180,E1 -6079.299,E2 -6079.299} C_VEL
LIN {X 0,Y 496.718,Z 447.342,A -85,B 0,C 180,E1 -6080.102,E2 -6080.102} C_VEL
LIN {X 0,Y 496.377,Z 457.881,A -85,B 0,C 180,E1 -6081.043,E2 -6081.043} C_VEL
LIN {X 0,Y 496.048,Z 467.234,A -85,B 0,C 180,E1 -6082.082,E2 -6082.082} C_VEL
LIN {X 0,Y 495.77,Z 475.484,A -85,B 0,C 180,E1 -6083.207,E2 -6083.207} C_VEL
LIN {X 0,Y 495.486,Z 482.84,A -85,B 0,C 180,E1 -6084.441,E2 -6084.441} C_VEL
LIN {X 0,Y 495.308,Z 489.675,A -85,B 0,C 180,E1 -6085.912,E2 -6085.912} C_VEL
LIN {X 0,Y 495.173,Z 494.734,A -85,B 0,C 180,E1 -6087.362,E2 -6087.362} C_VEL
LIN {X 0,Y 495.098,Z 497.403,A -85,B 0,C 180,E1 -6088.386,E2 -6088.386} C_VEL
LIN {X 0,Y 494.969,Z 500.247,A -85,B 0,C 180,E1 -6089.999,E2 -6089.999} C_VEL
LIN {X 0,Y 494.935,Z 501.472,A -85,B 0,C 180,E1 -6091.676,E2 -6091.676} C_VEL
LIN {X 0,Y 494.957,Z 500.974,A -85,B 0,C 180,E1 -6093.436,E2 -6093.436} C_VEL
LIN {X 0,Y 495.025,Z 499.29,A -85,B 0,C 180,E1 -6094.792,E2 -6094.792} C_VEL
LIN {X 0,Y 495.154,Z 496.469,A -85,B 0,C 180,E1 -6096.14,E2 -6096.14} C_VEL
LIN {X 0,Y 495.242,Z 492.489,A -85,B 0,C 180,E1 -6097.471,E2 -6097.471} C_VEL
LIN {X 0,Y 495.376,Z 487.246,A -85,B 0,C 180,E1 -6098.791,E2 -6098.791} C_VEL
LIN {X 0,Y 495.626,Z 480.558,A -85,B 0,C 180,E1 -6100.104,E2 -6100.104} C_VEL
LIN {X 0,Y 495.868,Z 472.335,A -85,B 0,C 180,E1 -6101.376,E2 -6101.376} C_VEL
LIN {X 0,Y 496.251,Z 463.442,A -85,B 0,C 180,E1 -6102.486,E2 -6102.486} C_VEL
LIN {X 0,Y 496.539,Z 453.964,A -85,B 0,C 180,E1 -6103.451,E2 -6103.451} C_VEL
LIN {X 0,Y 496.958,Z 443.29,A -85,B 0,C 180,E1 -6104.321,E2 -6104.321} C_VEL
LIN {X 0,Y 497.243,Z 432.09,A -85,B 0,C 180,E1 -6105.052,E2 -6105.052} C_VEL
LIN {X 0,Y 497.53,Z 420.529,A -85,B 0,C 180,E1 -6105.636,E2 -6105.636} C_VEL
LIN {X 0,Y 497.732,Z 407.924,A -85,B 0,C 180,E1 -6106.098,E2 -6106.098} C_VEL
LIN {X 0,Y 497.946,Z 395.445,A -85,B 0,C 180,E1 -6106.392,E2 -6106.392} C_VEL
LIN {X 0,Y 498.51,Z 302.334,A -85,B 0,C 180,E1 -6107.816,E2 -6107.816} C_VEL
LIN {X 0,Y 496.226,Z 290.605,A -85,B 0,C 180,E1 -6108.095,E2 -6108.095} C_VEL
LIN {X 0,Y 496.004,Z 279.93,A -85,B 0,C 180,E1 -6109.799,E2 -6109.799} C_VEL
LIN {X 0,Y 495.785,Z 278.73,A -85,B 0,C 180,E1 -6110,E2 -6110} C_VEL
LIN {X 0,Y 495.832,Z 278.726,A -85,B 0,C 180,E1 -6112.778,E2 -6112.778} C_VEL
LIN {X 0,Y 495.784,Z 278.733,A -85,B 0,C 180,E1 -6115.121,E2 -6115.121} C_VEL
LIN {X 0,Y 495.936,Z 278.709,A -85,B 0,C 180,E1 -6117.564,E2 -6117.564} C_VEL
LIN {X 0,Y 495.933,Z 278.706,A -85,B 0,C 180,E1 -6120,E2 -6120} C_VEL
LIN {X 0,Y 495.937,Z 278.708,A -85,B 0,C 180,E1 -6122.437,E2 -6122.437} C_VEL
LIN {X 0,Y 495.845,Z 278.717,A -85,B 0,C 180,E1 -6125.694,E2 -6125.694} C_VEL
LIN {X 0,Y 495.815,Z 278.72,A -85,B 0,C 180,E1 -6128.149,E2 -6128.149} C_VEL
LIN {X 0,Y 495.817,Z 278.723,A -85,B 0,C 180,E1 -6131.446,E2 -6131.446} C_VEL
LIN {X 0,Y 495.744,Z 278.734,A -85,B 0,C 180,E1 -6134.785,E2 -6134.785} C_VEL
LIN {X 0,Y 495.733,Z 278.733,A -85,B 0,C 180,E1 -6137.321,E2 -6137.321} C_VEL
LIN {X 0,Y 495.718,Z 278.73,A -85,B 0,C 180,E1 -6139.893,E2 -6139.893} C_VEL
LIN {X 0,Y 495.709,Z 278.738,A -85,B 0,C 180,E1 -6142.864,E2 -6142.864} C_VEL
LIN {X 0,Y 495.75,Z 278.726,A -85,B 0,C 180,E1 -6146.071,E2 -6146.071} C_VEL
LIN {X 0,Y 495.725,Z 278.735,A -85,B 0,C 180,E1 -6148.818,E2 -6148.818} C_VEL
LIN {X 0,Y 495.713,Z 278.733,A -85,B 0,C 180,E1 -6151.729,E2 -6151.729} C_VEL
LIN {X 0,Y 495.734,Z 278.731,A -85,B 0,C 180,E1 -6154.699,E2 -6154.699} C_VEL
LIN {X 0,Y 495.692,Z 278.739,A -85,B 0,C 180,E1 -6157.565,E2 -6157.565} C_VEL
LIN {X 0,Y 495.747,Z 278.73,A -85,B 0,C 180,E1 -6160.702,E2 -6160.702} C_VEL
LIN {X 0,Y 495.702,Z 278.734,A -85,B 0,C 180,E1 -6164.005,E2 -6164.005} C_VEL
LIN {X 0,Y 495.697,Z 278.74,A -85,B 0,C 180,E1 -6167.121,E2 -6167.121} C_VEL
LIN {X 0,Y 495.732,Z 278.731,A -85,B 0,C 180,E1 -6169.957,E2 -6169.957} C_VEL
LIN {X 0,Y 495.703,Z 278.735,A -85,B 0,C 180,E1 -6172.558,E2 -6172.558} C_VEL
LIN {X 0,Y 495.757,Z 278.737,A -85,B 0,C 180,E1 -6175.461,E2 -6175.461} C_VEL
LIN {X 0,Y 495.737,Z 278.735,A -85,B 0,C 180,E1 -6178.368,E2 -6178.368} C_VEL
LIN {X 0,Y 495.742,Z 278.737,A -85,B 0,C 180,E1 -6181.517,E2 -6181.517} C_VEL
LIN {X 0,Y 495.848,Z 278.92,A -85,B 0,C 180,E1 -6184.447,E2 -6184.447} C_VEL
LIN {X 0,Y 497.315,Z 287.547,A -85,B 0,C 180,E1 -6185.81,E2 -6185.81} C_VEL
LIN {X 0,Y 497.053,Z 303.675,A -85,B 0,C 180,E1 -6188.217,E2 -6188.217} C_VEL
LIN {X 0,Y 496.567,Z 324.643,A -85,B 0,C 180,E1 -6191.315,E2 -6191.315} C_VEL
LIN {X 0,Y 496.206,Z 342.578,A -85,B 0,C 180,E1 -6193.956,E2 -6193.956} C_VEL
LIN {X 0,Y 498.446,Z 360.329,A -85,B 0,C 180,E1 -6194.305,E2 -6194.305} C_VEL
LIN {X 0,Y 497.76,Z 451.801,A -85,B 0,C 180,E1 -6195.698,E2 -6195.698} C_VEL
LIN {X 0,Y 497.465,Z 465.018,A -85,B 0,C 180,E1 -6196.054,E2 -6196.054} C_VEL
LIN {X 0,Y 497.129,Z 477.788,A -85,B 0,C 180,E1 -6196.565,E2 -6196.565} C_VEL
LIN {X 0,Y 496.78,Z 490.429,A -85,B 0,C 180,E1 -6197.261,E2 -6197.261} C_VEL
LIN {X 0,Y 496.389,Z 501.599,A -85,B 0,C 180,E1 -6198.052,E2 -6198.052} C_VEL
LIN {X 0,Y 496.034,Z 512.088,A -85,B 0,C 180,E1 -6198.975,E2 -6198.975} C_VEL
LIN {X 0,Y 495.722,Z 521.514,A -85,B 0,C 180,E1 -6200.001,E2 -6200.001} C_VEL
LIN {X 0,Y 495.434,Z 530.66,A -85,B 0,C 180,E1 -6201.231,E2 -6201.231} C_VEL
LIN {X 0,Y 495.244,Z 538.032,A -85,B 0,C 180,E1 -6202.459,E2 -6202.459} C_VEL
LIN {X 0,Y 495.119,Z 544.241,A -85,B 0,C 180,E1 -6203.764,E2 -6203.764} C_VEL
LIN {X 0,Y 495.037,Z 549.193,A -85,B 0,C 180,E1 -6205.115,E2 -6205.115} C_VEL
LIN {X 0,Y 495.065,Z 551.549,A -85,B 0,C 180,E1 -6205.931,E2 -6205.931} C_VEL
LIN {X 0,Y 495.046,Z 553.461,A -85,B 0,C 180,E1 -6206.746,E2 -6206.746} C_VEL
LIN {X 0,Y 495.053,Z 554.895,A -85,B 0,C 180,E1 -6207.561,E2 -6207.561} C_VEL
LIN {X 0,Y 494.917,Z 556.547,A -85,B 0,C 180,E1 -6209.188,E2 -6209.188} C_VEL
LIN {X 0,Y 494.912,Z 556.778,A -85,B 0,C 180,E1 -6210.001,E2 -6210.001} C_VEL
LIN {X 0,Y 494.963,Z 555.96,A -85,B 0,C 180,E1 -6211.628,E2 -6211.628} C_VEL
LIN {X 0,Y 495.054,Z 554.962,A -85,B 0,C 180,E1 -6212.442,E2 -6212.442} C_VEL
LIN {X 0,Y 495.046,Z 553.545,A -85,B 0,C 180,E1 -6213.256,E2 -6213.256} C_VEL
LIN {X 0,Y 495.011,Z 550.567,A -85,B 0,C 180,E1 -6214.479,E2 -6214.479} C_VEL
LIN {X 0,Y 495.134,Z 546.539,A -85,B 0,C 180,E1 -6215.703,E2 -6215.703} C_VEL
LIN {X 0,Y 495.254,Z 540.325,A -85,B 0,C 180,E1 -6217.133,E2 -6217.133} C_VEL
LIN {X 0,Y 495.383,Z 533.539,A -85,B 0,C 180,E1 -6218.362,E2 -6218.362} C_VEL
LIN {X 0,Y 495.605,Z 525.12,A -85,B 0,C 180,E1 -6219.592,E2 -6219.592} C_VEL
LIN {X 0,Y 495.958,Z 516.454,A -85,B 0,C 180,E1 -6220.616,E2 -6220.616} C_VEL
LIN {X 0,Y 496.303,Z 506.956,A -85,B 0,C 180,E1 -6221.538,E2 -6221.538} C_VEL
LIN {X 0,Y 496.623,Z 495.289,A -85,B 0,C 180,E1 -6222.455,E2 -6222.455} C_VEL
LIN {X 0,Y 497.014,Z 483.454,A -85,B 0,C 180,E1 -6223.18,E2 -6223.18} C_VEL
LIN {X 0,Y 497.35,Z 471.294,A -85,B 0,C 180,E1 -6223.743,E2 -6223.743} C_VEL
LIN {X 0,Y 497.695,Z 458.104,A -85,B 0,C 180,E1 -6224.177,E2 -6224.177} C_VEL
LIN {X 0,Y 497.907,Z 445.365,A -85,B 0,C 180,E1 -6224.431,E2 -6224.431} C_VEL
LIN {X 0,Y 498.35,Z 358.256,A -85,B 0,C 180,E1 -6225.74,E2 -6225.74} C_VEL
LIN {X 0,Y 496.263,Z 343.598,A -85,B 0,C 180,E1 -6226.036,E2 -6226.036} C_VEL
LIN {X 0,Y 496.845,Z 324.367,A -85,B 0,C 180,E1 -6228.986,E2 -6228.986} C_VEL
LIN {X 0,Y 497.422,Z 305.085,A -85,B 0,C 180,E1 -6231.987,E2 -6231.987} C_VEL
LIN {X 0,Y 497.936,Z 289.905,A -85,B 0,C 180,E1 -6234.382,E2 -6234.382} C_VEL
LIN {X 0,Y 495.737,Z 278.737,A -85,B 0,C 180,E1 -6236.317,E2 -6236.317} C_VEL
LIN {X 0,Y 495.738,Z 278.736,A -85,B 0,C 180,E1 -6238.815,E2 -6238.815} C_VEL
LIN {X 0,Y 495.747,Z 278.729,A -85,B 0,C 180,E1 -6241.723,E2 -6241.723} C_VEL
LIN {X 0,Y 495.75,Z 278.736,A -85,B 0,C 180,E1 -6244.69,E2 -6244.69} C_VEL
LIN {X 0,Y 495.696,Z 278.734,A -85,B 0,C 180,E1 -6247.562,E2 -6247.562} C_VEL
LIN {X 0,Y 495.717,Z 278.74,A -85,B 0,C 180,E1 -6250.702,E2 -6250.702} C_VEL
LIN {X 0,Y 495.707,Z 278.734,A -85,B 0,C 180,E1 -6254,E2 -6254} C_VEL
LIN {X 0,Y 495.686,Z 278.739,A -85,B 0,C 180,E1 -6257.112,E2 -6257.112} C_VEL
LIN {X 0,Y 495.723,Z 278.735,A -85,B 0,C 180,E1 -6260.358,E2 -6260.358} C_VEL
LIN {X 0,Y 495.692,Z 278.736,A -85,B 0,C 180,E1 -6263.453,E2 -6263.453} C_VEL
LIN {X 0,Y 495.716,Z 278.736,A -85,B 0,C 180,E1 -6266.432,E2 -6266.432} C_VEL
LIN {X 0,Y 495.722,Z 278.733,A -85,B 0,C 180,E1 -6269.31,E2 -6269.31} C_VEL
LIN {X 0,Y 495.743,Z 278.731,A -85,B 0,C 180,E1 -6272.106,E2 -6272.106} C_VEL
LIN {X 0,Y 495.697,Z 278.743,A -85,B 0,C 180,E1 -6274.827,E2 -6274.827} C_VEL
LIN {X 0,Y 495.714,Z 278.734,A -85,B 0,C 180,E1 -6277.493,E2 -6277.493} C_VEL
LIN {X 0,Y 495.727,Z 278.733,A -85,B 0,C 180,E1 -6280.107,E2 -6280.107} C_VEL
LIN {X 0,Y 495.722,Z 278.737,A -85,B 0,C 180,E1 -6282.679,E2 -6282.679} C_VEL
LIN {X 0,Y 495.747,Z 278.732,A -85,B 0,C 180,E1 -6285.215,E2 -6285.215} C_VEL
LIN {X 0,Y 495.834,Z 278.722,A -85,B 0,C 180,E1 -6288.554,E2 -6288.554} C_VEL
LIN {X 0,Y 495.835,Z 278.718,A -85,B 0,C 180,E1 -6291.851,E2 -6291.851} C_VEL
LIN {X 0,Y 495.85,Z 278.719,A -85,B 0,C 180,E1 -6294.306,E2 -6294.306} C_VEL
LIN {X 0,Y 495.952,Z 278.704,A -85,B 0,C 180,E1 -6297.563,E2 -6297.563} C_VEL
LIN {X 0,Y 495.953,Z 278.704,A -85,B 0,C 180,E1 -6300,E2 -6300} C_VEL
LIN {X 0,Y 495.952,Z 278.708,A -85,B 0,C 180,E1 -6302.436,E2 -6302.436} C_VEL
LIN {X 0,Y 495.851,Z 278.717,A -85,B 0,C 180,E1 -6305.694,E2 -6305.694} C_VEL
LIN {X 0,Y 495.836,Z 278.719,A -85,B 0,C 180,E1 -6308.148,E2 -6308.148} C_VEL
LIN {X 0,Y 495.837,Z 278.72,A -85,B 0,C 180,E1 -6311.445,E2 -6311.445} C_VEL
LIN {X 0,Y 495.753,Z 278.733,A -85,B 0,C 180,E1 -6314.784,E2 -6314.784} C_VEL
LIN {X 0,Y 495.75,Z 278.732,A -85,B 0,C 180,E1 -6317.319,E2 -6317.319} C_VEL
LIN {X 0,Y 495.736,Z 278.731,A -85,B 0,C 180,E1 -6319.891,E2 -6319.891} C_VEL
LIN {X 0,Y 495.727,Z 278.737,A -85,B 0,C 180,E1 -6322.862,E2 -6322.862} C_VEL
LIN {X 0,Y 495.759,Z 278.729,A -85,B 0,C 180,E1 -6326.069,E2 -6326.069} C_VEL
LIN {X 0,Y 495.75,Z 278.734,A -85,B 0,C 180,E1 -6328.816,E2 -6328.816} C_VEL
LIN {X 0,Y 495.73,Z 278.732,A -85,B 0,C 180,E1 -6331.727,E2 -6331.727} C_VEL
LIN {X 0,Y 495.75,Z 278.734,A -85,B 0,C 180,E1 -6334.697,E2 -6334.697} C_VEL
LIN {X 0,Y 495.706,Z 278.736,A -85,B 0,C 180,E1 -6337.563,E2 -6337.563} C_VEL
LIN {X 0,Y 495.758,Z 278.734,A -85,B 0,C 180,E1 -6340.7,E2 -6340.7} C_VEL
LIN {X 0,Y 495.713,Z 278.734,A -85,B 0,C 180,E1 -6344.003,E2 -6344.003} C_VEL
LIN {X 0,Y 495.746,Z 278.734,A -85,B 0,C 180,E1 -6347.123,E2 -6347.123} C_VEL
LIN {X 0,Y 495.775,Z 278.728,A -85,B 0,C 180,E1 -6350.367,E2 -6350.367} C_VEL
LIN {X 0,Y 495.721,Z 278.735,A -85,B 0,C 180,E1 -6353.458,E2 -6353.458} C_VEL
LIN {X 0,Y 495.748,Z 278.731,A -85,B 0,C 180,E1 -6356.437,E2 -6356.437} C_VEL
LIN {X 0,Y 495.741,Z 278.734,A -85,B 0,C 180,E1 -6359.314,E2 -6359.314} C_VEL
LIN {X 0,Y 495.744,Z 278.731,A -85,B 0,C 180,E1 -6360.785,E2 -6360.785} C_VEL
LIN {X 0,Y 495.089,Z 278.815,A -85,B 0,C 180,E1 -6361.464,E2 -6361.464} C_VEL
LIN {X 0,Y 492.232,Z 279.17,A -85,B 0,C 180,E1 -6362.566,E2 -6362.566} C_VEL
LIN {X 0,Y 489.822,Z 279.471,A -85,B 0,C 180,E1 -6363.455,E2 -6363.455} C_VEL
LIN {X 0,Y 488.807,Z 279.595,A -85,B 0,C 180,E1 -6364.141,E2 -6364.141} C_VEL
LIN {X 0,Y 488.736,Z 279.604,A -85,B 0,C 180,E1 -6364.374,E2 -6364.374} C_VEL
LIN {X 0,Y 488.716,Z 279.609,A -85,B 0,C 180,E1 -6367.154,E2 -6367.154} C_VEL
LIN {X 0,Y 488.72,Z 279.605,A -85,B 0,C 180,E1 -6369.811,E2 -6369.811} C_VEL
LIN {X 0,Y 488.73,Z 279.605,A -85,B 0,C 180,E1 -6372.424,E2 -6372.424} C_VEL
LIN {X 0,Y 488.758,Z 279.605,A -85,B 0,C 180,E1 -6375,E2 -6375} C_VEL
LIN {X 0,Y 488.803,Z 279.595,A -85,B 0,C 180,E1 -6378.387,E2 -6378.387} C_VEL
LIN {X 0,Y 488.815,Z 279.594,A -85,B 0,C 180,E1 -6381.733,E2 -6381.733} C_VEL
LIN {X 0,Y 488.852,Z 279.588,A -85,B 0,C 180,E1 -6384.223,E2 -6384.223} C_VEL
LIN {X 0,Y 488.959,Z 279.578,A -85,B 0,C 180,E1 -6387.528,E2 -6387.528} C_VEL
LIN {X 0,Y 488.951,Z 279.581,A -85,B 0,C 180,E1 -6390.822,E2 -6390.822} C_VEL
LIN {X 0,Y 488.959,Z 279.576,A -85,B 0,C 180,E1 -6392.47,E2 -6392.47} C_VEL
LIN {X 0,Y 488.844,Z 279.59,A -85,B 0,C 180,E1 -6395.774,E2 -6395.774} C_VEL
LIN {X 0,Y 488.812,Z 279.593,A -85,B 0,C 180,E1 -6398.264,E2 -6398.264} C_VEL
LIN {X 0,Y 488.825,Z 279.593,A -85,B 0,C 180,E1 -6401.609,E2 -6401.609} C_VEL
LIN {X 0,Y 488.753,Z 279.607,A -85,B 0,C 180,E1 -6404.998,E2 -6404.998} C_VEL
LIN {X 0,Y 488.744,Z 279.602,A -85,B 0,C 180,E1 -6408.439,E2 -6408.439} C_VEL
LIN {X 0,Y 488.728,Z 279.61,A -85,B 0,C 180,E1 -6411.066,E2 -6411.066} C_VEL
LIN {X 0,Y 488.686,Z 279.61,A -85,B 0,C 180,E1 -6413.742,E2 -6413.742} C_VEL
LIN {X 0,Y 488.781,Z 279.601,A -85,B 0,C 180,E1 -6416.942,E2 -6416.942} C_VEL
LIN {X 0,Y 488.698,Z 279.606,A -85,B 0,C 180,E1 -6420.361,E2 -6420.361} C_VEL
LIN {X 0,Y 488.712,Z 279.608,A -85,B 0,C 180,E1 -6423.481,E2 -6423.481} C_VEL
LIN {X 0,Y 488.664,Z 279.61,A -85,B 0,C 180,E1 -6426.352,E2 -6426.352} C_VEL
LIN {X 0,Y 488.721,Z 279.611,A -85,B 0,C 180,E1 -6429.246,E2 -6429.246} C_VEL
LIN {X 0,Y 488.722,Z 279.608,A -85,B 0,C 180,E1 -6432.515,E2 -6432.515} C_VEL
LIN {X 0,Y 488.815,Z 279.784,A -85,B 0,C 180,E1 -6433.357,E2 -6433.357} C_VEL
LIN {X 0,Y 489.413,Z 284.473,A -85,B 0,C 180,E1 -6434.355,E2 -6434.355} C_VEL
LIN {X 0,Y 489.257,Z 291.598,A -85,B 0,C 180,E1 -6435.813,E2 -6435.813} C_VEL
LIN {X 0,Y 491.759,Z 304.053,A -85,B 0,C 180,E1 -6436.095,E2 -6436.095} C_VEL
LIN {X 0,Y 491.013,Z 398.816,A -85,B 0,C 180,E1 -6437.567,E2 -6437.567} C_VEL
LIN {X 0,Y 490.848,Z 411.846,A -85,B 0,C 180,E1 -6437.934,E2 -6437.934} C_VEL
LIN {X 0,Y 490.53,Z 423.717,A -85,B 0,C 180,E1 -6438.42,E2 -6438.42} C_VEL
LIN {X 0,Y 490.194,Z 435.348,A -85,B 0,C 180,E1 -6439.057,E2 -6439.057} C_VEL
LIN {X 0,Y 489.832,Z 445.743,A -85,B 0,C 180,E1 -6439.786,E2 -6439.786} C_VEL
LIN {X 0,Y 489.478,Z 456.081,A -85,B 0,C 180,E1 -6440.688,E2 -6440.688} C_VEL
LIN {X 0,Y 489.139,Z 465.631,A -85,B 0,C 180,E1 -6441.712,E2 -6441.712} C_VEL
LIN {X 0,Y 488.794,Z 474.297,A -85,B 0,C 180,E1 -6442.852,E2 -6442.852} C_VEL
LIN {X 0,Y 488.52,Z 481.964,A -85,B 0,C 180,E1 -6444.11,E2 -6444.11} C_VEL
LIN {X 0,Y 488.288,Z 488.596,A -85,B 0,C 180,E1 -6445.477,E2 -6445.477} C_VEL
LIN {X 0,Y 488.138,Z 493.692,A -85,B 0,C 180,E1 -6446.832,E2 -6446.832} C_VEL
LIN {X 0,Y 488.048,Z 497.396,A -85,B 0,C 180,E1 -6448.158,E2 -6448.158} C_VEL
LIN {X 0,Y 487.888,Z 500.294,A -85,B 0,C 180,E1 -6449.724,E2 -6449.724} C_VEL
LIN {X 0,Y 487.859,Z 501.364,A -85,B 0,C 180,E1 -6450.673,E2 -6450.673} C_VEL
LIN {X 0,Y 487.848,Z 501.855,A -85,B 0,C 180,E1 -6451.615,E2 -6451.615} C_VEL
LIN {X 0,Y 487.87,Z 501.522,A -85,B 0,C 180,E1 -6453.256,E2 -6453.256} C_VEL
LIN {X 0,Y 487.921,Z 500.333,A -85,B 0,C 180,E1 -6454.398,E2 -6454.398} C_VEL
LIN {X 0,Y 488.017,Z 497.888,A -85,B 0,C 180,E1 -6455.768,E2 -6455.768} C_VEL
LIN {X 0,Y 488.163,Z 494.287,A -85,B 0,C 180,E1 -6457.126,E2 -6457.126} C_VEL
LIN {X 0,Y 488.29,Z 489.46,A -85,B 0,C 180,E1 -6458.468,E2 -6458.468} C_VEL
LIN {X 0,Y 488.527,Z 483.202,A -85,B 0,C 180,E1 -6459.802,E2 -6459.802} C_VEL
LIN {X 0,Y 488.772,Z 475.381,A -85,B 0,C 180,E1 -6461.124,E2 -6461.124} C_VEL
LIN {X 0,Y 489.119,Z 467.321,A -85,B 0,C 180,E1 -6462.222,E2 -6462.222} C_VEL
LIN {X 0,Y 489.475,Z 457.427,A -85,B 0,C 180,E1 -6463.312,E2 -6463.312} C_VEL
LIN {X 0,Y 489.928,Z 446.335,A -85,B 0,C 180,E1 -6464.291,E2 -6464.291} C_VEL
LIN {X 0,Y 490.247,Z 435.608,A -85,B 0,C 180,E1 -6465.047,E2 -6465.047} C_VEL
LIN {X 0,Y 490.56,Z 423.76,A -85,B 0,C 180,E1 -6465.693,E2 -6465.693} C_VEL
LIN {X 0,Y 490.832,Z 410.318,A -85,B 0,C 180,E1 -6466.23,E2 -6466.23} C_VEL
LIN {X 0,Y 491.044,Z 397.201,A -85,B 0,C 180,E1 -6466.567,E2 -6466.567} C_VEL
LIN {X 0,Y 491.828,Z 303.957,A -85,B 0,C 180,E1 -6468.022,E2 -6468.022} C_VEL
LIN {X 0,Y 489.29,Z 290.979,A -85,B 0,C 180,E1 -6468.34,E2 -6468.34} C_VEL
LIN {X 0,Y 489.082,Z 281.427,A -85,B 0,C 180,E1 -6469.862,E2 -6469.862} C_VEL
LIN {X 0,Y 488.746,Z 279.607,A -85,B 0,C 180,E1 -6470.169,E2 -6470.169} C_VEL
LIN {X 0,Y 488.804,Z 279.601,A -85,B 0,C 180,E1 -6472.727,E2 -6472.727} C_VEL
LIN {X 0,Y 488.754,Z 279.609,A -85,B 0,C 180,E1 -6475.051,E2 -6475.051} C_VEL
LIN {X 0,Y 488.905,Z 279.585,A -85,B 0,C 180,E1 -6477.529,E2 -6477.529} C_VEL
LIN {X 0,Y 488.905,Z 279.582,A -85,B 0,C 180,E1 -6480,E2 -6480} C_VEL
LIN {X 0,Y 488.906,Z 279.584,A -85,B 0,C 180,E1 -6482.472,E2 -6482.472} C_VEL
LIN {X 0,Y 488.803,Z 279.594,A -85,B 0,C 180,E1 -6485.777,E2 -6485.777} C_VEL
LIN {X 0,Y 488.761,Z 279.599,A -85,B 0,C 180,E1 -6488.268,E2 -6488.268} C_VEL
LIN {X 0,Y 488.777,Z 279.598,A -85,B 0,C 180,E1 -6491.614,E2 -6491.614} C_VEL
LIN {X 0,Y 488.713,Z 279.61,A -85,B 0,C 180,E1 -6495.002,E2 -6495.002} C_VEL
LIN {X 0,Y 488.702,Z 279.606,A -85,B 0,C 180,E1 -6498.445,E2 -6498.445} C_VEL
LIN {X 0,Y 488.654,Z 279.617,A -85,B 0,C 180,E1 -6501.073,E2 -6501.073} C_VEL
LIN {X 0,Y 488.641,Z 279.614,A -85,B 0,C 180,E1 -6503.749,E2 -6503.749} C_VEL
LIN {X 0,Y 488.751,Z 279.604,A -85,B 0,C 180,E1 -6506.948,E2 -6506.948} C_VEL
LIN {X 0,Y 488.664,Z 279.611,A -85,B 0,C 180,E1 -6510.366,E2 -6510.366} C_VEL
LIN {X 0,Y 488.693,Z 279.61,A -85,B 0,C 180,E1 -6513.488,E2 -6513.488} C_VEL
LIN {X 0,Y 488.647,Z 279.613,A -85,B 0,C 180,E1 -6516.359,E2 -6516.359} C_VEL
LIN {X 0,Y 488.711,Z 279.61,A -85,B 0,C 180,E1 -6519.254,E2 -6519.254} C_VEL
LIN {X 0,Y 488.658,Z 279.61,A -85,B 0,C 180,E1 -6522.53,E2 -6522.53} C_VEL
LIN {X 0,Y 488.681,Z 279.615,A -85,B 0,C 180,E1 -6525.203,E2 -6525.203} C_VEL
LIN {X 0,Y 488.68,Z 279.609,A -85,B 0,C 180,E1 -6528.404,E2 -6528.404} C_VEL
LIN {X 0,Y 488.678,Z 279.613,A -85,B 0,C 180,E1 -6530.952,E2 -6530.952} C_VEL
LIN {X 0,Y 488.655,Z 279.616,A -85,B 0,C 180,E1 -6533.872,E2 -6533.872} C_VEL
LIN {X 0,Y 488.72,Z 279.611,A -85,B 0,C 180,E1 -6536.881,E2 -6536.881} C_VEL
LIN {X 0,Y 488.708,Z 279.613,A -85,B 0,C 180,E1 -6539.785,E2 -6539.785} C_VEL
LIN {X 0,Y 488.713,Z 279.611,A -85,B 0,C 180,E1 -6543.076,E2 -6543.076} C_VEL
LIN {X 0,Y 488.807,Z 279.812,A -85,B 0,C 180,E1 -6544.281,E2 -6544.281} C_VEL
LIN {X 0,Y 490.333,Z 288.449,A -85,B 0,C 180,E1 -6545.669,E2 -6545.669} C_VEL
LIN {X 0,Y 490.204,Z 298.77,A -85,B 0,C 180,E1 -6547.23,E2 -6547.23} C_VEL
LIN {X 0,Y 489.733,Z 317.741,A -85,B 0,C 180,E1 -6550.076,E2 -6550.076} C_VEL
LIN {X 0,Y 489.333,Z 336.495,A -85,B 0,C 180,E1 -6552.88,E2 -6552.88} C_VEL
LIN {X 0,Y 489.2,Z 342.076,A -85,B 0,C 180,E1 -6553.713,E2 -6553.713} C_VEL
LIN {X 0,Y 491.586,Z 360.85,A -85,B 0,C 180,E1 -6554.095,E2 -6554.095} C_VEL
LIN {X 0,Y 490.862,Z 452.169,A -85,B 0,C 180,E1 -6555.519,E2 -6555.519} C_VEL
LIN {X 0,Y 490.522,Z 465.869,A -85,B 0,C 180,E1 -6555.906,E2 -6555.906} C_VEL
LIN {X 0,Y 490.176,Z 478.279,A -85,B 0,C 180,E1 -6556.424,E2 -6556.424} C_VEL
LIN {X 0,Y 489.81,Z 489.896,A -85,B 0,C 180,E1 -6557.079,E2 -6557.079} C_VEL
LIN {X 0,Y 489.418,Z 501.068,A -85,B 0,C 180,E1 -6557.879,E2 -6557.879} C_VEL
LIN {X 0,Y 489.044,Z 511.584,A -85,B 0,C 180,E1 -6558.816,E2 -6558.816} C_VEL
LIN {X 0,Y 488.692,Z 521.032,A -85,B 0,C 180,E1 -6559.856,E2 -6559.856} C_VEL
LIN {X 0,Y 488.373,Z 530.191,A -85,B 0,C 180,E1 -6561.103,E2 -6561.103} C_VEL
LIN {X 0,Y 488.178,Z 537.578,A -85,B 0,C 180,E1 -6562.35,E2 -6562.35} C_VEL
LIN {X 0,Y 488.047,Z 543.185,A -85,B 0,C 180,E1 -6563.525,E2 -6563.525} C_VEL
LIN {X 0,Y 488.043,Z 547.421,A -85,B 0,C 180,E1 -6564.631,E2 -6564.631} C_VEL
LIN {X 0,Y 487.96,Z 551.13,A -85,B 0,C 180,E1 -6565.872,E2 -6565.872} C_VEL
LIN {X 0,Y 487.97,Z 553.05,A -85,B 0,C 180,E1 -6566.699,E2 -6566.699} C_VEL
LIN {X 0,Y 487.959,Z 554.491,A -85,B 0,C 180,E1 -6567.525,E2 -6567.525} C_VEL
LIN {X 0,Y 487.893,Z 555.518,A -85,B 0,C 180,E1 -6568.351,E2 -6568.351} C_VEL
LIN {X 0,Y 487.84,Z 556.151,A -85,B 0,C 180,E1 -6569.176,E2 -6569.176} C_VEL
LIN {X 0,Y 487.832,Z 556.383,A -85,B 0,C 180,E1 -6570.001,E2 -6570.001} C_VEL
LIN {X 0,Y 487.893,Z 555.568,A -85,B 0,C 180,E1 -6571.652,E2 -6571.652} C_VEL
LIN {X 0,Y 487.959,Z 554.568,A -85,B 0,C 180,E1 -6572.478,E2 -6572.478} C_VEL
LIN {X 0,Y 487.97,Z 553.149,A -85,B 0,C 180,E1 -6573.304,E2 -6573.304} C_VEL
LIN {X 0,Y 487.923,Z 550.167,A -85,B 0,C 180,E1 -6574.545,E2 -6574.545} C_VEL
LIN {X 0,Y 488.028,Z 546.13,A -85,B 0,C 180,E1 -6575.786,E2 -6575.786} C_VEL
LIN {X 0,Y 488.179,Z 539.906,A -85,B 0,C 180,E1 -6577.237,E2 -6577.237} C_VEL
LIN {X 0,Y 488.325,Z 533.11,A -85,B 0,C 180,E1 -6578.484,E2 -6578.484} C_VEL
LIN {X 0,Y 488.554,Z 524.673,A -85,B 0,C 180,E1 -6579.732,E2 -6579.732} C_VEL
LIN {X 0,Y 488.922,Z 515.98,A -85,B 0,C 180,E1 -6580.77,E2 -6580.77} C_VEL
LIN {X 0,Y 489.294,Z 505.267,A -85,B 0,C 180,E1 -6581.811,E2 -6581.811} C_VEL
LIN {X 0,Y 489.671,Z 493.831,A -85,B 0,C 180,E1 -6582.701,E2 -6582.701} C_VEL
LIN {X 0,Y 490.072,Z 482.841,A -85,B 0,C 180,E1 -6583.37,E2 -6583.37} C_VEL
LIN {X 0,Y 490.423,Z 470.602,A -85,B 0,C 180,E1 -6583.941,E2 -6583.941} C_VEL
LIN {X 0,Y 490.79,Z 457.283,A -85,B 0,C 180,E1 -6584.38,E2 -6584.38} C_VEL
LIN {X 0,Y 491.023,Z 442.428,A -85,B 0,C 180,E1 -6584.664,E2 -6584.664} C_VEL
LIN {X 0,Y 491.468,Z 358.695,A -85,B 0,C 180,E1 -6585.95,E2 -6585.95} C_VEL
LIN {X 0,Y 489.28,Z 343.235,A -85,B 0,C 180,E1 -6586.269,E2 -6586.269} C_VEL
LIN {X 0,Y 489.85,Z 324.017,A -85,B 0,C 180,E1 -6589.267,E2 -6589.267} C_VEL
LIN {X 0,Y 490.533,Z 304.733,A -85,B 0,C 180,E1 -6592.312,E2 -6592.312} C_VEL
LIN {X 0,Y 490.976,Z 290.929,A -85,B 0,C 180,E1 -6594.525,E2 -6594.525} C_VEL
LIN {X 0,Y 488.723,Z 279.61,A -85,B 0,C 180,E1 -6596.509,E2 -6596.509} C_VEL
LIN {X 0,Y 488.704,Z 279.607,A -85,B 0,C 180,E1 -6599.27,E2 -6599.27} C_VEL
LIN {X 0,Y 488.69,Z 279.611,A -85,B 0,C 180,E1 -6602.146,E2 -6602.146} C_VEL
LIN {X 0,Y 488.703,Z 279.608,A -85,B 0,C 180,E1 -6605.114,E2 -6605.114} C_VEL
LIN {X 0,Y 488.647,Z 279.615,A -85,B 0,C 180,E1 -6608.2,E2 -6608.2} C_VEL
LIN {X 0,Y 488.681,Z 279.612,A -85,B 0,C 180,E1 -6610.339,E2 -6610.339} C_VEL
LIN {X 0,Y 488.659,Z 279.611,A -85,B 0,C 180,E1 -6613.654,E2 -6613.654} C_VEL
LIN {X 0,Y 488.658,Z 279.615,A -85,B 0,C 180,E1 -6616.342,E2 -6616.342} C_VEL
LIN {X 0,Y 488.685,Z 279.608,A -85,B 0,C 180,E1 -6619.671,E2 -6619.671} C_VEL
LIN {X 0,Y 488.644,Z 279.62,A -85,B 0,C 180,E1 -6622.837,E2 -6622.837} C_VEL
LIN {X 0,Y 488.694,Z 279.608,A -85,B 0,C 180,E1 -6625.884,E2 -6625.884} C_VEL
LIN {X 0,Y 488.663,Z 279.618,A -85,B 0,C 180,E1 -6628.818,E2 -6628.818} C_VEL
LIN {X 0,Y 488.712,Z 279.605,A -85,B 0,C 180,E1 -6631.669,E2 -6631.669} C_VEL
LIN {X 0,Y 488.674,Z 279.614,A -85,B 0,C 180,E1 -6634.44,E2 -6634.44} C_VEL
LIN {X 0,Y 488.688,Z 279.612,A -85,B 0,C 180,E1 -6637.151,E2 -6637.151} C_VEL
LIN {X 0,Y 488.686,Z 279.609,A -85,B 0,C 180,E1 -6639.808,E2 -6639.808} C_VEL
LIN {X 0,Y 488.675,Z 279.613,A -85,B 0,C 180,E1 -6642.421,E2 -6642.421} C_VEL
LIN {X 0,Y 488.722,Z 279.61,A -85,B 0,C 180,E1 -6644.998,E2 -6644.998} C_VEL
LIN {X 0,Y 488.789,Z 279.599,A -85,B 0,C 180,E1 -6648.387,E2 -6648.387} C_VEL
LIN {X 0,Y 488.78,Z 279.597,A -85,B 0,C 180,E1 -6651.733,E2 -6651.733} C_VEL
LIN {X 0,Y 488.809,Z 279.596,A -85,B 0,C 180,E1 -6654.223,E2 -6654.223} C_VEL
LIN {X 0,Y 488.92,Z 279.581,A -85,B 0,C 180,E1 -6657.528,E2 -6657.528} C_VEL
LIN {X 0,Y 488.925,Z 279.58,A -85,B 0,C 180,E1 -6660,E2 -6660} C_VEL
LIN {X 0,Y 488.921,Z 279.584,A -85,B 0,C 180,E1 -6662.471,E2 -6662.471} C_VEL
LIN {X 0,Y 488.809,Z 279.594,A -85,B 0,C 180,E1 -6665.776,E2 -6665.776} C_VEL
LIN {X 0,Y 488.781,Z 279.599,A -85,B 0,C 180,E1 -6668.267,E2 -6668.267} C_VEL
LIN {X 0,Y 488.797,Z 279.596,A -85,B 0,C 180,E1 -6671.612,E2 -6671.612} C_VEL
LIN {X 0,Y 488.725,Z 279.609,A -85,B 0,C 180,E1 -6675.001,E2 -6675.001} C_VEL
LIN {X 0,Y 488.721,Z 279.608,A -85,B 0,C 180,E1 -6678.443,E2 -6678.443} C_VEL
LIN {X 0,Y 488.673,Z 279.616,A -85,B 0,C 180,E1 -6681.072,E2 -6681.072} C_VEL
LIN {X 0,Y 488.659,Z 279.613,A -85,B 0,C 180,E1 -6683.747,E2 -6683.747} C_VEL
LIN {X 0,Y 488.761,Z 279.604,A -85,B 0,C 180,E1 -6686.945,E2 -6686.945} C_VEL
LIN {X 0,Y 488.704,Z 279.608,A -85,B 0,C 180,E1 -6690.22,E2 -6690.22} C_VEL
LIN {X 0,Y 488.709,Z 279.608,A -85,B 0,C 180,E1 -6693.486,E2 -6693.486} C_VEL
LIN {X 0,Y 488.663,Z 279.614,A -85,B 0,C 180,E1 -6696.357,E2 -6696.357} C_VEL
LIN {X 0,Y 488.724,Z 279.609,A -85,B 0,C 180,E1 -6699.251,E2 -6699.251} C_VEL
LIN {X 0,Y 488.67,Z 279.615,A -85,B 0,C 180,E1 -6702.527,E2 -6702.527} C_VEL
LIN {X 0,Y 488.692,Z 279.613,A -85,B 0,C 180,E1 -6705.2,E2 -6705.2} C_VEL
LIN {X 0,Y 488.718,Z 279.608,A -85,B 0,C 180,E1 -6707.481,E2 -6707.481} C_VEL
LIN {X 0,Y 488.733,Z 279.609,A -85,B 0,C 180,E1 -6710.752,E2 -6710.752} C_VEL
LIN {X 0,Y 488.672,Z 279.611,A -85,B 0,C 180,E1 -6713.87,E2 -6713.87} C_VEL
LIN {X 0,Y 488.727,Z 279.609,A -85,B 0,C 180,E1 -6716.879,E2 -6716.879} C_VEL
LIN {X 0,Y 488.713,Z 279.606,A -85,B 0,C 180,E1 -6719.782,E2 -6719.782} C_VEL
LIN {X 0,Y 488.784,Z 279.601,A -85,B 0,C 180,E1 -6723.057,E2 -6723.057} C_VEL
LIN {X 0,Y 488.736,Z 279.604,A -85,B 0,C 180,E1 -6724.374,E2 -6724.374} C_VEL
LIN {X 0,Y 488.092,Z 279.689,A -85,B 0,C 180,E1 -6725.062,E2 -6725.062} C_VEL
LIN {X 0,Y 485.222,Z 280.045,A -85,B 0,C 180,E1 -6726.178,E2 -6726.178} C_VEL
LIN {X 0,Y 482.774,Z 280.35,A -85,B 0,C 180,E1 -6727.078,E2 -6727.078} C_VEL
LIN {X 0,Y 481.716,Z 280.478,A -85,B 0,C 180,E1 -6727.773,E2 -6727.773} C_VEL
LIN {X 0,Y 481.629,Z 280.489,A -85,B 0,C 180,E1 -6728.009,E2 -6728.009} C_VEL
LIN {X 0,Y 481.701,Z 280.481,A -85,B 0,C 180,E1 -6730.393,E2 -6730.393} C_VEL
LIN {X 0,Y 481.687,Z 280.486,A -85,B 0,C 180,E1 -6733.034,E2 -6733.034} C_VEL
LIN {X 0,Y 481.686,Z 280.483,A -85,B 0,C 180,E1 -6735.639,E2 -6735.639} C_VEL
LIN {X 0,Y 481.748,Z 280.474,A -85,B 0,C 180,E1 -6738.215,E2 -6738.215} C_VEL
LIN {X 0,Y 481.761,Z 280.474,A -85,B 0,C 180,E1 -6741.611,E2 -6741.611} C_VEL
LIN {X 0,Y 481.813,Z 280.465,A -85,B 0,C 180,E1 -6744.139,E2 -6744.139} C_VEL
LIN {X 0,Y 481.926,Z 280.454,A -85,B 0,C 180,E1 -6747.491,E2 -6747.491} C_VEL
LIN {X 0,Y 481.902,Z 280.459,A -85,B 0,C 180,E1 -6750.834,E2 -6750.834} C_VEL
LIN {X 0,Y 481.926,Z 280.452,A -85,B 0,C 180,E1 -6752.506,E2 -6752.506} C_VEL
LIN {X 0,Y 481.804,Z 280.466,A -85,B 0,C 180,E1 -6755.859,E2 -6755.859} C_VEL
LIN {X 0,Y 481.757,Z 280.472,A -85,B 0,C 180,E1 -6758.386,E2 -6758.386} C_VEL
LIN {X 0,Y 481.788,Z 280.469,A -85,B 0,C 180,E1 -6761.781,E2 -6761.781} C_VEL
LIN {X 0,Y 481.734,Z 280.48,A -85,B 0,C 180,E1 -6765.222,E2 -6765.222} C_VEL
LIN {X 0,Y 481.701,Z 280.481,A -85,B 0,C 180,E1 -6768.719,E2 -6768.719} C_VEL
LIN {X 0,Y 481.659,Z 280.487,A -85,B 0,C 180,E1 -6771.39,E2 -6771.39} C_VEL
LIN {X 0,Y 481.667,Z 280.482,A -85,B 0,C 180,E1 -6774.11,E2 -6774.11} C_VEL
LIN {X 0,Y 481.734,Z 280.482,A -85,B 0,C 180,E1 -6777.137,E2 -6777.137} C_VEL
LIN {X 0,Y 481.668,Z 280.484,A -85,B 0,C 180,E1 -6779.737,E2 -6779.737} C_VEL
LIN {X 0,Y 481.651,Z 280.486,A -85,B 0,C 180,E1 -6782.67,E2 -6782.67} C_VEL
LIN {X 0,Y 481.618,Z 280.49,A -85,B 0,C 180,E1 -6785.705,E2 -6785.705} C_VEL
LIN {X 0,Y 481.694,Z 280.486,A -85,B 0,C 180,E1 -6789.351,E2 -6789.351} C_VEL
LIN {X 0,Y 481.655,Z 280.488,A -85,B 0,C 180,E1 -6792.153,E2 -6792.153} C_VEL
LIN {X 0,Y 481.75,Z 280.612,A -85,B 0,C 180,E1 -6793.207,E2 -6793.207} C_VEL
LIN {X 0,Y 482.417,Z 285.991,A -85,B 0,C 180,E1 -6794.362,E2 -6794.362} C_VEL
LIN {X 0,Y 482.31,Z 291.878,A -85,B 0,C 180,E1 -6795.574,E2 -6795.574} C_VEL
LIN {X 0,Y 484.968,Z 305.25,A -85,B 0,C 180,E1 -6795.887,E2 -6795.887} C_VEL
LIN {X 0,Y 484.145,Z 398.628,A -85,B 0,C 180,E1 -6797.358,E2 -6797.358} C_VEL
LIN {X 0,Y 483.951,Z 412.187,A -85,B 0,C 180,E1 -6797.743,E2 -6797.743} C_VEL
LIN {X 0,Y 483.628,Z 424.609,A -85,B 0,C 180,E1 -6798.262,E2 -6798.262} C_VEL
LIN {X 0,Y 483.245,Z 436.217,A -85,B 0,C 180,E1 -6798.916,E2 -6798.916} C_VEL
LIN {X 0,Y 482.81,Z 447.856,A -85,B 0,C 180,E1 -6799.764,E2 -6799.764} C_VEL
LIN {X 0,Y 482.418,Z 458.368,A -85,B 0,C 180,E1 -6800.724,E2 -6800.724} C_VEL
LIN {X 0,Y 482.048,Z 468.007,A -85,B 0,C 180,E1 -6801.821,E2 -6801.821} C_VEL
LIN {X 0,Y 481.71,Z 476.412,A -85,B 0,C 180,E1 -6803,E2 -6803} C_VEL
LIN {X 0,Y 481.417,Z 483.764,A -85,B 0,C 180,E1 -6804.272,E2 -6804.272} C_VEL
LIN {X 0,Y 481.199,Z 490.569,A -85,B 0,C 180,E1 -6805.786,E2 -6805.786} C_VEL
LIN {X 0,Y 481.044,Z 495.615,A -85,B 0,C 180,E1 -6807.278,E2 -6807.278} C_VEL
LIN {X 0,Y 480.953,Z 498.111,A -85,B 0,C 180,E1 -6808.261,E2 -6808.261} C_VEL
LIN {X 0,Y 480.808,Z 500.52,A -85,B 0,C 180,E1 -6809.575,E2 -6809.575} C_VEL
LIN {X 0,Y 480.77,Z 502.145,A -85,B 0,C 180,E1 -6811.28,E2 -6811.28} C_VEL
LIN {X 0,Y 480.755,Z 502.334,A -85,B 0,C 180,E1 -6812.109,E2 -6812.109} C_VEL
LIN {X 0,Y 480.773,Z 502.033,A -85,B 0,C 180,E1 -6813.074,E2 -6813.074} C_VEL
LIN {X 0,Y 480.816,Z 501.296,A -85,B 0,C 180,E1 -6813.992,E2 -6813.992} C_VEL
LIN {X 0,Y 480.894,Z 499.952,A -85,B 0,C 180,E1 -6814.956,E2 -6814.956} C_VEL
LIN {X 0,Y 481.017,Z 497.148,A -85,B 0,C 180,E1 -6816.31,E2 -6816.31} C_VEL
LIN {X 0,Y 481.118,Z 493.127,A -85,B 0,C 180,E1 -6817.679,E2 -6817.679} C_VEL
LIN {X 0,Y 481.31,Z 487.425,A -85,B 0,C 180,E1 -6819.131,E2 -6819.131} C_VEL
LIN {X 0,Y 481.578,Z 481.051,A -85,B 0,C 180,E1 -6820.388,E2 -6820.388} C_VEL
LIN {X 0,Y 481.85,Z 473.79,A -85,B 0,C 180,E1 -6821.548,E2 -6821.548} C_VEL
LIN {X 0,Y 482.201,Z 465.645,A -85,B 0,C 180,E1 -6822.616,E2 -6822.616} C_VEL
LIN {X 0,Y 482.584,Z 456.081,A -85,B 0,C 180,E1 -6823.644,E2 -6823.644} C_VEL
LIN {X 0,Y 483.025,Z 446.359,A -85,B 0,C 180,E1 -6824.493,E2 -6824.493} C_VEL
LIN {X 0,Y 483.343,Z 435.542,A -85,B 0,C 180,E1 -6825.259,E2 -6825.259} C_VEL
LIN {X 0,Y 483.698,Z 423.551,A -85,B 0,C 180,E1 -6825.915,E2 -6825.915} C_VEL
LIN {X 0,Y 483.956,Z 410.747,A -85,B 0,C 180,E1 -6826.431,E2 -6826.431} C_VEL
LIN {X 0,Y 484.171,Z 397.796,A -85,B 0,C 180,E1 -6826.771,E2 -6826.771} C_VEL
LIN {X 0,Y 485.027,Z 304.676,A -85,B 0,C 180,E1 -6828.257,E2 -6828.257} C_VEL
LIN {X 0,Y 482.352,Z 291.283,A -85,B 0,C 180,E1 -6828.603,E2 -6828.603} C_VEL
LIN {X 0,Y 482.2,Z 283.001,A -85,B 0,C 180,E1 -6829.928,E2 -6829.928} C_VEL
LIN {X 0,Y 481.704,Z 280.485,A -85,B 0,C 180,E1 -6830.368,E2 -6830.368} C_VEL
LIN {X 0,Y 481.715,Z 280.483,A -85,B 0,C 180,E1 -6833.298,E2 -6833.298} C_VEL
LIN {X 0,Y 481.609,Z 280.494,A -85,B 0,C 180,E1 -6835.816,E2 -6835.816} C_VEL
LIN {X 0,Y 481.873,Z 280.462,A -85,B 0,C 180,E1 -6837.493,E2 -6837.493} C_VEL
LIN {X 0,Y 481.877,Z 280.457,A -85,B 0,C 180,E1 -6840,E2 -6840} C_VEL
LIN {X 0,Y 481.874,Z 280.461,A -85,B 0,C 180,E1 -6842.508,E2 -6842.508} C_VEL
LIN {X 0,Y 481.763,Z 280.471,A -85,B 0,C 180,E1 -6845.861,E2 -6845.861} C_VEL
LIN {X 0,Y 481.707,Z 280.479,A -85,B 0,C 180,E1 -6848.39,E2 -6848.39} C_VEL
LIN {X 0,Y 481.741,Z 280.474,A -85,B 0,C 180,E1 -6851.786,E2 -6851.786} C_VEL
LIN {X 0,Y 481.692,Z 280.484,A -85,B 0,C 180,E1 -6855.226,E2 -6855.226} C_VEL
LIN {X 0,Y 481.659,Z 280.485,A -85,B 0,C 180,E1 -6858.724,E2 -6858.724} C_VEL
LIN {X 0,Y 481.593,Z 280.495,A -85,B 0,C 180,E1 -6861.398,E2 -6861.398} C_VEL
LIN {X 0,Y 481.626,Z 280.487,A -85,B 0,C 180,E1 -6864.116,E2 -6864.116} C_VEL
LIN {X 0,Y 481.704,Z 280.485,A -85,B 0,C 180,E1 -6867.143,E2 -6867.143} C_VEL
LIN {X 0,Y 481.633,Z 280.488,A -85,B 0,C 180,E1 -6869.745,E2 -6869.745} C_VEL
LIN {X 0,Y 481.63,Z 280.488,A -85,B 0,C 180,E1 -6872.678,E2 -6872.678} C_VEL
LIN {X 0,Y 481.601,Z 280.493,A -85,B 0,C 180,E1 -6875.713,E2 -6875.713} C_VEL
LIN {X 0,Y 481.682,Z 280.485,A -85,B 0,C 180,E1 -6879.358,E2 -6879.358} C_VEL
LIN {X 0,Y 481.62,Z 280.486,A -85,B 0,C 180,E1 -6882.164,E2 -6882.164} C_VEL
LIN {X 0,Y 481.63,Z 280.492,A -85,B 0,C 180,E1 -6885.547,E2 -6885.547} C_VEL
LIN {X 0,Y 481.63,Z 280.492,A -85,B 0,C 180,E1 -6888.962,E2 -6888.962} C_VEL
LIN {X 0,Y 481.63,Z 280.488,A -85,B 0,C 180,E1 -6891.997,E2 -6891.997} C_VEL
LIN {X 0,Y 481.668,Z 280.492,A -85,B 0,C 180,E1 -6895.322,E2 -6895.322} C_VEL
LIN {X 0,Y 481.627,Z 280.493,A -85,B 0,C 180,E1 -6898.315,E2 -6898.315} C_VEL
LIN {X 0,Y 481.662,Z 280.492,A -85,B 0,C 180,E1 -6901.221,E2 -6901.221} C_VEL
LIN {X 0,Y 481.735,Z 280.663,A -85,B 0,C 180,E1 -6904.094,E2 -6904.094} C_VEL
LIN {X 0,Y 483.339,Z 289.364,A -85,B 0,C 180,E1 -6905.522,E2 -6905.522} C_VEL
LIN {X 0,Y 483.328,Z 298.215,A -85,B 0,C 180,E1 -6906.887,E2 -6906.887} C_VEL
LIN {X 0,Y 482.73,Z 318.689,A -85,B 0,C 180,E1 -6909.997,E2 -6909.997} C_VEL
LIN {X 0,Y 482.299,Z 337.494,A -85,B 0,C 180,E1 -6912.841,E2 -6912.841} C_VEL
LIN {X 0,Y 482.23,Z 341.693,A -85,B 0,C 180,E1 -6913.463,E2 -6913.463} C_VEL
LIN {X 0,Y 484.772,Z 360.82,A -85,B 0,C 180,E1 -6913.865,E2 -6913.865} C_VEL
LIN {X 0,Y 483.971,Z 451.4,A -85,B 0,C 180,E1 -6915.308,E2 -6915.308} C_VEL
LIN {X 0,Y 483.623,Z 465.197,A -85,B 0,C 180,E1 -6915.7,E2 -6915.7} C_VEL
LIN {X 0,Y 483.234,Z 477.676,A -85,B 0,C 180,E1 -6916.225,E2 -6916.225} C_VEL
LIN {X 0,Y 482.841,Z 489.336,A -85,B 0,C 180,E1 -6916.889,E2 -6916.889} C_VEL
LIN {X 0,Y 482.447,Z 500.449,A -85,B 0,C 180,E1 -6917.694,E2 -6917.694} C_VEL
LIN {X 0,Y 482.052,Z 511.08,A -85,B 0,C 180,E1 -6918.651,E2 -6918.651} C_VEL
LIN {X 0,Y 481.656,Z 520.552,A -85,B 0,C 180,E1 -6919.706,E2 -6919.706} C_VEL
LIN {X 0,Y 481.321,Z 529.73,A -85,B 0,C 180,E1 -6920.971,E2 -6920.971} C_VEL
LIN {X 0,Y 481.09,Z 537.133,A -85,B 0,C 180,E1 -6922.236,E2 -6922.236} C_VEL
LIN {X 0,Y 480.945,Z 543.283,A -85,B 0,C 180,E1 -6923.556,E2 -6923.556} C_VEL
LIN {X 0,Y 480.902,Z 548.354,A -85,B 0,C 180,E1 -6924.971,E2 -6924.971} C_VEL
LIN {X 0,Y 480.858,Z 550.716,A -85,B 0,C 180,E1 -6925.811,E2 -6925.811} C_VEL
LIN {X 0,Y 480.895,Z 552.644,A -85,B 0,C 180,E1 -6926.65,E2 -6926.65} C_VEL
LIN {X 0,Y 480.869,Z 554.088,A -85,B 0,C 180,E1 -6927.489,E2 -6927.489} C_VEL
LIN {X 0,Y 480.824,Z 555.12,A -85,B 0,C 180,E1 -6928.326,E2 -6928.326} C_VEL
LIN {X 0,Y 480.765,Z 555.754,A -85,B 0,C 180,E1 -6929.164,E2 -6929.164} C_VEL
LIN {X 0,Y 480.755,Z 555.988,A -85,B 0,C 180,E1 -6930.001,E2 -6930.001} C_VEL
LIN {X 0,Y 480.825,Z 555.174,A -85,B 0,C 180,E1 -6931.676,E2 -6931.676} C_VEL
LIN {X 0,Y 480.869,Z 554.171,A -85,B 0,C 180,E1 -6932.514,E2 -6932.514} C_VEL
LIN {X 0,Y 480.895,Z 552.749,A -85,B 0,C 180,E1 -6933.352,E2 -6933.352} C_VEL
LIN {X 0,Y 480.841,Z 549.76,A -85,B 0,C 180,E1 -6934.612,E2 -6934.612} C_VEL
LIN {X 0,Y 480.93,Z 545.712,A -85,B 0,C 180,E1 -6935.872,E2 -6935.872} C_VEL
LIN {X 0,Y 481.1,Z 539.47,A -85,B 0,C 180,E1 -6937.344,E2 -6937.344} C_VEL
LIN {X 0,Y 481.265,Z 532.656,A -85,B 0,C 180,E1 -6938.609,E2 -6938.609} C_VEL
LIN {X 0,Y 481.493,Z 524.188,A -85,B 0,C 180,E1 -6939.876,E2 -6939.876} C_VEL
LIN {X 0,Y 481.891,Z 515.467,A -85,B 0,C 180,E1 -6940.929,E2 -6940.929} C_VEL
LIN {X 0,Y 482.254,Z 504.931,A -85,B 0,C 180,E1 -6941.967,E2 -6941.967} C_VEL
LIN {X 0,Y 482.665,Z 494.351,A -85,B 0,C 180,E1 -6942.808,E2 -6942.808} C_VEL
LIN {X 0,Y 483.125,Z 482.187,A -85,B 0,C 180,E1 -6943.566,E2 -6943.566} C_VEL
LIN {X 0,Y 483.492,Z 469.867,A -85,B 0,C 180,E1 -6944.145,E2 -6944.145} C_VEL
LIN {X 0,Y 483.874,Z 457.339,A -85,B 0,C 180,E1 -6944.563,E2 -6944.563} C_VEL
LIN {X 0,Y 484.12,Z 444.626,A -85,B 0,C 180,E1 -6944.825,E2 -6944.825} C_VEL
LIN {X 0,Y 484.634,Z 359.482,A -85,B 0,C 180,E1 -6946.155,E2 -6946.155} C_VEL
LIN {X 0,Y 482.28,Z 342.891,A -85,B 0,C 180,E1 -6946.509,E2 -6946.509} C_VEL
LIN {X 0,Y 482.924,Z 323.644,A -85,B 0,C 180,E1 -6949.555,E2 -6949.555} C_VEL
LIN {X 0,Y 483.629,Z 304.362,A -85,B 0,C 180,E1 -6952.649,E2 -6952.649} C_VEL
LIN {X 0,Y 484.127,Z 293.345,A -85,B 0,C 180,E1 -6954.438,E2 -6954.438} C_VEL
LIN {X 0,Y 481.989,Z 282.138,A -85,B 0,C 180,E1 -6956.405,E2 -6956.405} C_VEL
LIN {X 0,Y 481.661,Z 280.49,A -85,B 0,C 180,E1 -6956.716,E2 -6956.716} C_VEL
LIN {X 0,Y 481.667,Z 280.483,A -85,B 0,C 180,E1 -6959.74,E2 -6959.74} C_VEL
LIN {X 0,Y 481.645,Z 280.493,A -85,B 0,C 180,E1 -6962.674,E2 -6962.674} C_VEL
LIN {X 0,Y 481.619,Z 280.488,A -85,B 0,C 180,E1 -6965.709,E2 -6965.709} C_VEL
LIN {X 0,Y 481.644,Z 280.49,A -85,B 0,C 180,E1 -6968.859,E2 -6968.859} C_VEL
LIN {X 0,Y 481.611,Z 280.491,A -85,B 0,C 180,E1 -6972.161,E2 -6972.161} C_VEL
LIN {X 0,Y 481.638,Z 280.486,A -85,B 0,C 180,E1 -6975.54,E2 -6975.54} C_VEL
LIN {X 0,Y 481.607,Z 280.495,A -85,B 0,C 180,E1 -6978.953,E2 -6978.953} C_VEL
LIN {X 0,Y 481.617,Z 280.49,A -85,B 0,C 180,E1 -6981.993,E2 -6981.993} C_VEL
LIN {X 0,Y 481.658,Z 280.485,A -85,B 0,C 180,E1 -6985.315,E2 -6985.315} C_VEL
LIN {X 0,Y 481.616,Z 280.492,A -85,B 0,C 180,E1 -6988.309,E2 -6988.309} C_VEL
LIN {X 0,Y 481.668,Z 280.485,A -85,B 0,C 180,E1 -6991.216,E2 -6991.216} C_VEL
LIN {X 0,Y 481.64,Z 280.487,A -85,B 0,C 180,E1 -6994.039,E2 -6994.039} C_VEL
LIN {X 0,Y 481.623,Z 280.495,A -85,B 0,C 180,E1 -6996.816,E2 -6996.816} C_VEL
LIN {X 0,Y 481.66,Z 280.485,A -85,B 0,C 180,E1 -6999.501,E2 -6999.501} C_VEL
LIN {X 0,Y 481.654,Z 280.486,A -85,B 0,C 180,E1 -7002.156,E2 -7002.156} C_VEL
LIN {X 0,Y 481.705,Z 280.484,A -85,B 0,C 180,E1 -7004.774,E2 -7004.774} C_VEL
LIN {X 0,Y 481.752,Z 280.475,A -85,B 0,C 180,E1 -7008.215,E2 -7008.215} C_VEL
LIN {X 0,Y 481.726,Z 280.476,A -85,B 0,C 180,E1 -7011.611,E2 -7011.611} C_VEL
LIN {X 0,Y 481.769,Z 280.472,A -85,B 0,C 180,E1 -7014.139,E2 -7014.139} C_VEL
LIN {X 0,Y 481.888,Z 280.457,A -85,B 0,C 180,E1 -7017.492,E2 -7017.492} C_VEL
LIN {X 0,Y 481.869,Z 280.463,A -85,B 0,C 180,E1 -7020.835,E2 -7020.835} C_VEL
LIN {X 0,Y 481.888,Z 280.459,A -85,B 0,C 180,E1 -7022.507,E2 -7022.507} C_VEL
LIN {X 0,Y 481.77,Z 280.471,A -85,B 0,C 180,E1 -7025.861,E2 -7025.861} C_VEL
LIN {X 0,Y 481.727,Z 280.479,A -85,B 0,C 180,E1 -7028.388,E2 -7028.388} C_VEL
LIN {X 0,Y 481.761,Z 280.472,A -85,B 0,C 180,E1 -7031.784,E2 -7031.784} C_VEL
LIN {X 0,Y 481.706,Z 280.483,A -85,B 0,C 180,E1 -7035.225,E2 -7035.225} C_VEL
LIN {X 0,Y 481.678,Z 280.486,A -85,B 0,C 180,E1 -7038.723,E2 -7038.723} C_VEL
LIN {X 0,Y 481.611,Z 280.493,A -85,B 0,C 180,E1 -7041.396,E2 -7041.396} C_VEL
LIN {X 0,Y 481.643,Z 280.487,A -85,B 0,C 180,E1 -7044.114,E2 -7044.114} C_VEL
LIN {X 0,Y 481.716,Z 280.482,A -85,B 0,C 180,E1 -7047.14,E2 -7047.14} C_VEL
LIN {X 0,Y 481.659,Z 280.485,A -85,B 0,C 180,E1 -7049.742,E2 -7049.742} C_VEL
LIN {X 0,Y 481.645,Z 280.491,A -85,B 0,C 180,E1 -7052.676,E2 -7052.676} C_VEL
LIN {X 0,Y 481.617,Z 280.491,A -85,B 0,C 180,E1 -7055.711,E2 -7055.711} C_VEL
LIN {X 0,Y 481.695,Z 280.484,A -85,B 0,C 180,E1 -7059.356,E2 -7059.356} C_VEL
LIN {X 0,Y 481.627,Z 280.489,A -85,B 0,C 180,E1 -7062.162,E2 -7062.162} C_VEL
LIN {X 0,Y 481.641,Z 280.489,A -85,B 0,C 180,E1 -7065.544,E2 -7065.544} C_VEL
LIN {X 0,Y 481.656,Z 280.486,A -85,B 0,C 180,E1 -7068.086,E2 -7068.086} C_VEL
LIN {X 0,Y 481.688,Z 280.485,A -85,B 0,C 180,E1 -7071.146,E2 -7071.146} C_VEL
LIN {X 0,Y 481.655,Z 280.49,A -85,B 0,C 180,E1 -7074.796,E2 -7074.796} C_VEL
LIN {X 0,Y 481.66,Z 280.488,A -85,B 0,C 180,E1 -7077.327,E2 -7077.327} C_VEL
LIN {X 0,Y 481.669,Z 280.484,A -85,B 0,C 180,E1 -7080.26,E2 -7080.26} C_VEL
LIN {X 0,Y 481.738,Z 280.479,A -85,B 0,C 180,E1 -7083.113,E2 -7083.113} C_VEL
LIN {X 0,Y 481.667,Z 280.484,A -85,B 0,C 180,E1 -7085.887,E2 -7085.887} C_VEL
LIN {X 0,Y 481.629,Z 280.489,A -85,B 0,C 180,E1 -7088.009,E2 -7088.009} C_VEL
LIN {X 0,Y 480.963,Z 280.576,A -85,B 0,C 180,E1 -7088.707,E2 -7088.707} C_VEL
LIN {X 0,Y 478.136,Z 280.926,A -85,B 0,C 180,E1 -7089.841,E2 -7089.841} C_VEL
LIN {X 0,Y 475.751,Z 281.226,A -85,B 0,C 180,E1 -7090.756,E2 -7090.756} C_VEL
LIN {X 0,Y 474.732,Z 281.35,A -85,B 0,C 180,E1 -7091.461,E2 -7091.461} C_VEL
LIN {X 0,Y 474.651,Z 281.358,A -85,B 0,C 180,E1 -7091.7,E2 -7091.7} C_VEL
LIN {X 0,Y 474.697,Z 281.354,A -85,B 0,C 180,E1 -7094.544,E2 -7094.544} C_VEL
LIN {X 0,Y 474.701,Z 281.351,A -85,B 0,C 180,E1 -7098.037,E2 -7098.037} C_VEL
LIN {X 0,Y 474.726,Z 281.351,A -85,B 0,C 180,E1 -7101.486,E2 -7101.486} C_VEL
LIN {X 0,Y 474.776,Z 281.342,A -85,B 0,C 180,E1 -7104.052,E2 -7104.052} C_VEL
LIN {X 0,Y 474.891,Z 281.33,A -85,B 0,C 180,E1 -7107.454,E2 -7107.454} C_VEL
LIN {X 0,Y 474.91,Z 281.325,A -85,B 0,C 180,E1 -7109.999,E2 -7109.999} C_VEL
LIN {X 0,Y 474.892,Z 281.329,A -85,B 0,C 180,E1 -7112.543,E2 -7112.543} C_VEL
LIN {X 0,Y 474.766,Z 281.343,A -85,B 0,C 180,E1 -7115.946,E2 -7115.946} C_VEL
LIN {X 0,Y 474.723,Z 281.349,A -85,B 0,C 180,E1 -7118.511,E2 -7118.511} C_VEL
LIN {X 0,Y 474.732,Z 281.347,A -85,B 0,C 180,E1 -7121.959,E2 -7121.959} C_VEL
LIN {X 0,Y 474.671,Z 281.355,A -85,B 0,C 180,E1 -7125.765,E2 -7125.765} C_VEL
LIN {X 0,Y 474.654,Z 281.363,A -85,B 0,C 180,E1 -7129.007,E2 -7129.007} C_VEL
LIN {X 0,Y 474.624,Z 281.361,A -85,B 0,C 180,E1 -7131.723,E2 -7131.723} C_VEL
LIN {X 0,Y 474.647,Z 281.358,A -85,B 0,C 180,E1 -7134.489,E2 -7134.489} C_VEL
LIN {X 0,Y 474.681,Z 281.358,A -85,B 0,C 180,E1 -7137.335,E2 -7137.335} C_VEL
LIN {X 0,Y 474.596,Z 281.366,A -85,B 0,C 180,E1 -7140.809,E2 -7140.809} C_VEL
LIN {X 0,Y 474.614,Z 281.361,A -85,B 0,C 180,E1 -7143.98,E2 -7143.98} C_VEL
LIN {X 0,Y 474.551,Z 281.372,A -85,B 0,C 180,E1 -7146.897,E2 -7146.897} C_VEL
LIN {X 0,Y 474.638,Z 281.363,A -85,B 0,C 180,E1 -7149.65,E2 -7149.65} C_VEL
LIN {X 0,Y 474.684,Z 281.437,A -85,B 0,C 180,E1 -7153.047,E2 -7153.047} C_VEL
LIN {X 0,Y 475.417,Z 285.802,A -85,B 0,C 180,E1 -7154.003,E2 -7154.003} C_VEL
LIN {X 0,Y 475.388,Z 292.397,A -85,B 0,C 180,E1 -7155.344,E2 -7155.344} C_VEL
LIN {X 0,Y 478.165,Z 306.828,A -85,B 0,C 180,E1 -7155.679,E2 -7155.679} C_VEL
LIN {X 0,Y 477.266,Z 400.062,A -85,B 0,C 180,E1 -7157.182,E2 -7157.182} C_VEL
LIN {X 0,Y 477.047,Z 412.531,A -85,B 0,C 180,E1 -7157.546,E2 -7157.546} C_VEL
LIN {X 0,Y 476.708,Z 425.233,A -85,B 0,C 180,E1 -7158.085,E2 -7158.085} C_VEL
LIN {X 0,Y 476.293,Z 437.545,A -85,B 0,C 180,E1 -7158.802,E2 -7158.802} C_VEL
LIN {X 0,Y 475.832,Z 449.453,A -85,B 0,C 180,E1 -7159.699,E2 -7159.699} C_VEL
LIN {X 0,Y 475.423,Z 459.677,A -85,B 0,C 180,E1 -7160.669,E2 -7160.669} C_VEL
LIN {X 0,Y 474.975,Z 469.783,A -85,B 0,C 180,E1 -7161.866,E2 -7161.866} C_VEL
LIN {X 0,Y 474.633,Z 478.08,A -85,B 0,C 180,E1 -7163.081,E2 -7163.081} C_VEL
LIN {X 0,Y 474.324,Z 485.288,A -85,B 0,C 180,E1 -7164.4,E2 -7164.4} C_VEL
LIN {X 0,Y 474.139,Z 491.011,A -85,B 0,C 180,E1 -7165.719,E2 -7165.719} C_VEL
LIN {X 0,Y 473.989,Z 496.057,A -85,B 0,C 180,E1 -7167.236,E2 -7167.236} C_VEL
LIN {X 0,Y 473.81,Z 499.568,A -85,B 0,C 180,E1 -7168.725,E2 -7168.725} C_VEL
LIN {X 0,Y 473.723,Z 501.13,A -85,B 0,C 180,E1 -7169.708,E2 -7169.708} C_VEL
LIN {X 0,Y 473.702,Z 502.419,A -85,B 0,C 180,E1 -7171.072,E2 -7171.072} C_VEL
LIN {X 0,Y 473.706,Z 502.546,A -85,B 0,C 180,E1 -7172.88,E2 -7172.88} C_VEL
LIN {X 0,Y 473.76,Z 501.074,A -85,B 0,C 180,E1 -7174.52,E2 -7174.52} C_VEL
LIN {X 0,Y 473.897,Z 498.586,A -85,B 0,C 180,E1 -7175.932,E2 -7175.932} C_VEL
LIN {X 0,Y 474.044,Z 494.946,A -85,B 0,C 180,E1 -7177.328,E2 -7177.328} C_VEL
LIN {X 0,Y 474.195,Z 490.214,A -85,B 0,C 180,E1 -7178.669,E2 -7178.669} C_VEL
LIN {X 0,Y 474.476,Z 483.728,A -85,B 0,C 180,E1 -7180.082,E2 -7180.082} C_VEL
LIN {X 0,Y 474.742,Z 476.62,A -85,B 0,C 180,E1 -7181.32,E2 -7181.32} C_VEL
LIN {X 0,Y 475.174,Z 467.7,A -85,B 0,C 180,E1 -7182.573,E2 -7182.573} C_VEL
LIN {X 0,Y 475.576,Z 457.708,A -85,B 0,C 180,E1 -7183.694,E2 -7183.694} C_VEL
LIN {X 0,Y 476.041,Z 447.847,A -85,B 0,C 180,E1 -7184.589,E2 -7184.589} C_VEL
LIN {X 0,Y 476.417,Z 437.287,A -85,B 0,C 180,E1 -7185.368,E2 -7185.368} C_VEL
LIN {X 0,Y 476.783,Z 425.761,A -85,B 0,C 180,E1 -7186.033,E2 -7186.033} C_VEL
LIN {X 0,Y 477.033,Z 412.939,A -85,B 0,C 180,E1 -7186.58,E2 -7186.58} C_VEL
LIN {X 0,Y 477.281,Z 400.184,A -85,B 0,C 180,E1 -7186.948,E2 -7186.948} C_VEL
LIN {X 0,Y 478.187,Z 305.218,A -85,B 0,C 180,E1 -7188.503,E2 -7188.503} C_VEL
LIN {X 0,Y 475.427,Z 291.638,A -85,B 0,C 180,E1 -7188.867,E2 -7188.867} C_VEL
LIN {X 0,Y 475.326,Z 284.648,A -85,B 0,C 180,E1 -7189.996,E2 -7189.996} C_VEL
LIN {X 0,Y 474.65,Z 281.364,A -85,B 0,C 180,E1 -7190.573,E2 -7190.573} C_VEL
LIN {X 0,Y 474.677,Z 281.361,A -85,B 0,C 180,E1 -7193.198,E2 -7193.198} C_VEL
LIN {X 0,Y 474.569,Z 281.372,A -85,B 0,C 180,E1 -7195.754,E2 -7195.754} C_VEL
LIN {X 0,Y 474.841,Z 281.338,A -85,B 0,C 180,E1 -7197.456,E2 -7197.456} C_VEL
LIN {X 0,Y 474.819,Z 281.343,A -85,B 0,C 180,E1 -7200.849,E2 -7200.849} C_VEL
LIN {X 0,Y 474.841,Z 281.337,A -85,B 0,C 180,E1 -7202.545,E2 -7202.545} C_VEL
LIN {X 0,Y 474.724,Z 281.348,A -85,B 0,C 180,E1 -7205.949,E2 -7205.949} C_VEL
LIN {X 0,Y 474.673,Z 281.356,A -85,B 0,C 180,E1 -7208.515,E2 -7208.515} C_VEL
LIN {X 0,Y 474.684,Z 281.353,A -85,B 0,C 180,E1 -7211.963,E2 -7211.963} C_VEL
LIN {X 0,Y 474.628,Z 281.36,A -85,B 0,C 180,E1 -7215.77,E2 -7215.77} C_VEL
LIN {X 0,Y 474.612,Z 281.367,A -85,B 0,C 180,E1 -7219.013,E2 -7219.013} C_VEL
LIN {X 0,Y 474.537,Z 281.371,A -85,B 0,C 180,E1 -7221.732,E2 -7221.732} C_VEL
LIN {X 0,Y 474.609,Z 281.363,A -85,B 0,C 180,E1 -7224.496,E2 -7224.496} C_VEL
LIN {X 0,Y 474.654,Z 281.361,A -85,B 0,C 180,E1 -7227.342,E2 -7227.342} C_VEL
LIN {X 0,Y 474.56,Z 281.372,A -85,B 0,C 180,E1 -7230.813,E2 -7230.813} C_VEL
LIN {X 0,Y 474.597,Z 281.362,A -85,B 0,C 180,E1 -7233.988,E2 -7233.988} C_VEL
LIN {X 0,Y 474.535,Z 281.375,A -85,B 0,C 180,E1 -7236.903,E2 -7236.903} C_VEL
LIN {X 0,Y 474.618,Z 281.363,A -85,B 0,C 180,E1 -7239.655,E2 -7239.655} C_VEL
LIN {X 0,Y 474.583,Z 281.367,A -85,B 0,C 180,E1 -7242.938,E2 -7242.938} C_VEL
LIN {X 0,Y 474.58,Z 281.367,A -85,B 0,C 180,E1 -7245.899,E2 -7245.899} C_VEL
LIN {X 0,Y 474.601,Z 281.368,A -85,B 0,C 180,E1 -7249.045,E2 -7249.045} C_VEL
LIN {X 0,Y 474.585,Z 281.368,A -85,B 0,C 180,E1 -7251.708,E2 -7251.708} C_VEL
LIN {X 0,Y 474.603,Z 281.367,A -85,B 0,C 180,E1 -7254.73,E2 -7254.73} C_VEL
LIN {X 0,Y 474.618,Z 281.37,A -85,B 0,C 180,E1 -7257.792,E2 -7257.792} C_VEL
LIN {X 0,Y 474.593,Z 281.371,A -85,B 0,C 180,E1 -7260.892,E2 -7260.892} C_VEL
LIN {X 0,Y 474.665,Z 281.424,A -85,B 0,C 180,E1 -7263.881,E2 -7263.881} C_VEL
LIN {X 0,Y 476.385,Z 290.384,A -85,B 0,C 180,E1 -7265.374,E2 -7265.374} C_VEL
LIN {X 0,Y 476.421,Z 297.773,A -85,B 0,C 180,E1 -7266.532,E2 -7266.532} C_VEL
LIN {X 0,Y 475.859,Z 316.826,A -85,B 0,C 180,E1 -7269.469,E2 -7269.469} C_VEL
LIN {X 0,Y 475.331,Z 337.072,A -85,B 0,C 180,E1 -7272.581,E2 -7272.581} C_VEL
LIN {X 0,Y 475.244,Z 341.052,A -85,B 0,C 180,E1 -7273.191,E2 -7273.191} C_VEL
LIN {X 0,Y 477.975,Z 361.907,A -85,B 0,C 180,E1 -7273.645,E2 -7273.645} C_VEL
LIN {X 0,Y 477.087,Z 450.976,A -85,B 0,C 180,E1 -7275.091,E2 -7275.091} C_VEL
LIN {X 0,Y 476.741,Z 464.722,A -85,B 0,C 180,E1 -7275.489,E2 -7275.489} C_VEL
LIN {X 0,Y 476.3,Z 477.177,A -85,B 0,C 180,E1 -7276.021,E2 -7276.021} C_VEL
LIN {X 0,Y 475.917,Z 488.353,A -85,B 0,C 180,E1 -7276.662,E2 -7276.662} C_VEL
LIN {X 0,Y 475.494,Z 499.219,A -85,B 0,C 180,E1 -7277.452,E2 -7277.452} C_VEL
LIN {X 0,Y 475.069,Z 509.484,A -85,B 0,C 180,E1 -7278.374,E2 -7278.374} C_VEL
LIN {X 0,Y 474.693,Z 518.306,A -85,B 0,C 180,E1 -7279.337,E2 -7279.337} C_VEL
LIN {X 0,Y 474.371,Z 526.438,A -85,B 0,C 180,E1 -7280.408,E2 -7280.408} C_VEL
LIN {X 0,Y 474.1,Z 534.4,A -85,B 0,C 180,E1 -7281.692,E2 -7281.692} C_VEL
LIN {X 0,Y 473.895,Z 541.704,A -85,B 0,C 180,E1 -7283.188,E2 -7283.188} C_VEL
LIN {X 0,Y 473.86,Z 546.58,A -85,B 0,C 180,E1 -7284.47,E2 -7284.47} C_VEL
LIN {X 0,Y 473.76,Z 550.307,A -85,B 0,C 180,E1 -7285.748,E2 -7285.748} C_VEL
LIN {X 0,Y 473.822,Z 552.24,A -85,B 0,C 180,E1 -7286.6,E2 -7286.6} C_VEL
LIN {X 0,Y 473.783,Z 553.687,A -85,B 0,C 180,E1 -7287.451,E2 -7287.451} C_VEL
LIN {X 0,Y 473.758,Z 554.722,A -85,B 0,C 180,E1 -7288.301,E2 -7288.301} C_VEL
LIN {X 0,Y 473.694,Z 555.359,A -85,B 0,C 180,E1 -7289.151,E2 -7289.151} C_VEL
LIN {X 0,Y 473.681,Z 555.593,A -85,B 0,C 180,E1 -7290.001,E2 -7290.001} C_VEL
LIN {X 0,Y 473.758,Z 554.776,A -85,B 0,C 180,E1 -7291.701,E2 -7291.701} C_VEL
LIN {X 0,Y 473.784,Z 553.77,A -85,B 0,C 180,E1 -7292.552,E2 -7292.552} C_VEL
LIN {X 0,Y 473.821,Z 552.343,A -85,B 0,C 180,E1 -7293.402,E2 -7293.402} C_VEL
LIN {X 0,Y 473.765,Z 549.346,A -85,B 0,C 180,E1 -7294.681,E2 -7294.681} C_VEL
LIN {X 0,Y 473.836,Z 545.286,A -85,B 0,C 180,E1 -7295.96,E2 -7295.96} C_VEL
LIN {X 0,Y 474.002,Z 539.027,A -85,B 0,C 180,E1 -7297.455,E2 -7297.455} C_VEL
LIN {X 0,Y 474.174,Z 532.195,A -85,B 0,C 180,E1 -7298.739,E2 -7298.739} C_VEL
LIN {X 0,Y 474.453,Z 523.704,A -85,B 0,C 180,E1 -7300.024,E2 -7300.024} C_VEL
LIN {X 0,Y 474.847,Z 514.954,A -85,B 0,C 180,E1 -7301.094,E2 -7301.094} C_VEL
LIN {X 0,Y 475.269,Z 504.628,A -85,B 0,C 180,E1 -7302.124,E2 -7302.124} C_VEL
LIN {X 0,Y 475.723,Z 493.484,A -85,B 0,C 180,E1 -7303.02,E2 -7303.02} C_VEL
LIN {X 0,Y 476.182,Z 481.532,A -85,B 0,C 180,E1 -7303.768,E2 -7303.768} C_VEL
LIN {X 0,Y 476.58,Z 469.139,A -85,B 0,C 180,E1 -7304.355,E2 -7304.355} C_VEL
LIN {X 0,Y 476.951,Z 456.463,A -85,B 0,C 180,E1 -7304.78,E2 -7304.78} C_VEL
LIN {X 0,Y 477.259,Z 441.619,A -85,B 0,C 180,E1 -7305.07,E2 -7305.07} C_VEL
LIN {X 0,Y 477.822,Z 360.348,A -85,B 0,C 180,E1 -7306.364,E2 -7306.364} C_VEL
LIN {X 0,Y 475.295,Z 342.487,A -85,B 0,C 180,E1 -7306.759,E2 -7306.759} C_VEL
LIN {X 0,Y 475.923,Z 324.767,A -85,B 0,C 180,E1 -7309.607,E2 -7309.607} C_VEL
LIN {X 0,Y 476.677,Z 305.366,A -85,B 0,C 180,E1 -7312.768,E2 -7312.768} C_VEL
LIN {X 0,Y 477.183,Z 294.327,A -85,B 0,C 180,E1 -7314.585,E2 -7314.585} C_VEL
LIN {X 0,Y 474.616,Z 281.373,A -85,B 0,C 180,E1 -7316.907,E2 -7316.907} C_VEL
LIN {X 0,Y 474.596,Z 281.368,A -85,B 0,C 180,E1 -7320.229,E2 -7320.229} C_VEL
LIN {X 0,Y 474.608,Z 281.363,A -85,B 0,C 180,E1 -7323.221,E2 -7323.221} C_VEL
LIN {X 0,Y 474.571,Z 281.37,A -85,B 0,C 180,E1 -7326.323,E2 -7326.323} C_VEL
LIN {X 0,Y 474.589,Z 281.364,A -85,B 0,C 180,E1 -7329.641,E2 -7329.641} C_VEL
LIN {X 0,Y 474.56,Z 281.372,A -85,B 0,C 180,E1 -7332.937,E2 -7332.937} C_VEL
LIN {X 0,Y 474.586,Z 281.365,A -85,B 0,C 180,E1 -7335.892,E2 -7335.892} C_VEL
LIN {X 0,Y 474.583,Z 281.369,A -85,B 0,C 180,E1 -7339.042,E2 -7339.042} C_VEL
LIN {X 0,Y 474.574,Z 281.366,A -85,B 0,C 180,E1 -7341.704,E2 -7341.704} C_VEL
LIN {X 0,Y 474.596,Z 281.37,A -85,B 0,C 180,E1 -7344.723,E2 -7344.723} C_VEL
LIN {X 0,Y 474.601,Z 281.363,A -85,B 0,C 180,E1 -7347.785,E2 -7347.785} C_VEL
LIN {X 0,Y 474.593,Z 281.37,A -85,B 0,C 180,E1 -7350.884,E2 -7350.884} C_VEL
LIN {X 0,Y 474.596,Z 281.364,A -85,B 0,C 180,E1 -7353.624,E2 -7353.624} C_VEL
LIN {X 0,Y 474.604,Z 281.367,A -85,B 0,C 180,E1 -7356.64,E2 -7356.64} C_VEL
LIN {X 0,Y 474.617,Z 281.363,A -85,B 0,C 180,E1 -7360.088,E2 -7360.088} C_VEL
LIN {X 0,Y 474.6,Z 281.369,A -85,B 0,C 180,E1 -7362.772,E2 -7362.772} C_VEL
LIN {X 0,Y 474.607,Z 281.364,A -85,B 0,C 180,E1 -7365.419,E2 -7365.419} C_VEL
LIN {X 0,Y 474.695,Z 281.353,A -85,B 0,C 180,E1 -7368.037,E2 -7368.037} C_VEL
LIN {X 0,Y 474.692,Z 281.353,A -85,B 0,C 180,E1 -7371.485,E2 -7371.485} C_VEL
LIN {X 0,Y 474.732,Z 281.348,A -85,B 0,C 180,E1 -7374.051,E2 -7374.051} C_VEL
LIN {X 0,Y 474.854,Z 281.334,A -85,B 0,C 180,E1 -7377.455,E2 -7377.455} C_VEL
LIN {X 0,Y 474.82,Z 281.341,A -85,B 0,C 180,E1 -7380.848,E2 -7380.848} C_VEL
LIN {X 0,Y 474.855,Z 281.335,A -85,B 0,C 180,E1 -7382.544,E2 -7382.544} C_VEL
LIN {X 0,Y 474.732,Z 281.348,A -85,B 0,C 180,E1 -7385.948,E2 -7385.948} C_VEL
LIN {X 0,Y 474.693,Z 281.356,A -85,B 0,C 180,E1 -7388.514,E2 -7388.514} C_VEL
LIN {X 0,Y 474.705,Z 281.352,A -85,B 0,C 180,E1 -7391.962,E2 -7391.962} C_VEL
LIN {X 0,Y 474.645,Z 281.359,A -85,B 0,C 180,E1 -7395.768,E2 -7395.768} C_VEL
LIN {X 0,Y 474.631,Z 281.364,A -85,B 0,C 180,E1 -7399.011,E2 -7399.011} C_VEL
LIN {X 0,Y 474.555,Z 281.37,A -85,B 0,C 180,E1 -7401.73,E2 -7401.73} C_VEL
LIN {X 0,Y 474.626,Z 281.365,A -85,B 0,C 180,E1 -7404.494,E2 -7404.494} C_VEL
LIN {X 0,Y 474.651,Z 281.361,A -85,B 0,C 180,E1 -7407.336,E2 -7407.336} C_VEL
LIN {X 0,Y 474.584,Z 281.368,A -85,B 0,C 180,E1 -7410.231,E2 -7410.231} C_VEL
LIN {X 0,Y 474.616,Z 281.367,A -85,B 0,C 180,E1 -7413.222,E2 -7413.222} C_VEL
LIN {X 0,Y 474.568,Z 281.37,A -85,B 0,C 180,E1 -7416.325,E2 -7416.325} C_VEL
LIN {X 0,Y 474.631,Z 281.361,A -85,B 0,C 180,E1 -7419.653,E2 -7419.653} C_VEL
LIN {X 0,Y 474.594,Z 281.368,A -85,B 0,C 180,E1 -7422.936,E2 -7422.936} C_VEL
LIN {X 0,Y 474.6,Z 281.365,A -85,B 0,C 180,E1 -7425.898,E2 -7425.898} C_VEL
LIN {X 0,Y 474.629,Z 281.364,A -85,B 0,C 180,E1 -7429.04,E2 -7429.04} C_VEL
LIN {X 0,Y 474.605,Z 281.364,A -85,B 0,C 180,E1 -7431.704,E2 -7431.704} C_VEL
LIN {X 0,Y 474.617,Z 281.367,A -85,B 0,C 180,E1 -7434.727,E2 -7434.727} C_VEL
LIN {X 0,Y 474.624,Z 281.362,A -85,B 0,C 180,E1 -7437.789,E2 -7437.789} C_VEL
